Universal Robots URScript: fai_chun_2024_v2.script

def fai_chun_2024_v2():
  set_tcp(p[0.0,0.0,0.0,0.0,0.0,0.0])
  set_gravity([0.0, 0.0, 9.82])
  set_target_payload(1.070000, [0.002000, 0.003000, 0.057000], [0.001723, 0.001723, 0.001723, 0.000000, 0.000000, 0.000000])
  set_tool_communication(True, 1000000, 2, 1, 1.5, 3.5)
  set_tool_output_mode(0)
  set_tool_digital_output_mode(0, 1)
  set_tool_digital_output_mode(1, 1)
  set_tool_voltage(0)
  step_count_453dca7f_7b0c_4a5f_b250_0e1aac3a1e4a = 0.0
  thread Step_Counter_Thread_f9e71c20_d700_42f0_a2ea_6ea405c4239a():
    while (True):
      step_count_453dca7f_7b0c_4a5f_b250_0e1aac3a1e4a = step_count_453dca7f_7b0c_4a5f_b250_0e1aac3a1e4a + 1.0
      sync()
    end
  end
  run Step_Counter_Thread_f9e71c20_d700_42f0_a2ea_6ea405c4239a()
  set_safety_mode_transition_hardness(1)
  set_standard_analog_input_domain(0, 1)
  set_standard_analog_input_domain(1, 1)
  set_tool_analog_input_domain(0, 1)
  set_tool_analog_input_domain(1, 1)
  set_analog_outputdomain(0, 0)
  set_analog_outputdomain(1, 0)
  set_input_actions_to_default()
  global Plane_1=p[-0.700006141123905,1.3454883874109249E-6,0.3910559577028425,-1.2089868272251132,-1.2089999932245832,1.20858562628424]
  global Plane_2=p[0.0,0.0,0.0,0.0,0.0,0.0]
  global Point_1=p[0.6913645118948067,-0.12399382748223003,0.49223711947071,-1.2983729986843258,1.1259514972191385,-1.2203503861141718]
  # begin: URCap Installation Node
  #   Source: External Control, 1.0.5, FZI Research Center for Information Technology
  #   Type: External Control
  # end: URCap Installation Node
  $ 1 "Robot Program"
  $ 2 "Script: test_first_drawing_8_m18.script"
  def Machining1():
    # Default parameters:
    global speed_ms = 0.3
    global speed_rads = 0.75
    global accel_mss = 3
    global accel_radss = 1.2
    global blend_radius_m = 0.001

    # Add subprograms here
    # Start of main program
    # Program generated by RoboDK v5.6.5 for UR10e on 02/02/2024 17:18:51
    # Using nominal kinematics.
    blend_radius_m = 0.001
    speed_ms = 1.000
    # set_reference(p[0.123734, -0.230000, -0.017586, 0.000000, 0.000000, 0.000000])
    set_tcp(p[0.000000, 0.000000, 0.252000, 0.000000, 0.000000, 0.000000])
    # Show Tool
    movej([-0.347318, -0.633716, -2.608659, -1.470014, 1.570796, 1.223478],accel_radss,speed_rads,0,blend_radius_m)
    movel([-0.347318, -0.633716, -2.608659, -1.470014, 1.570796, 1.223478],accel_mss,speed_ms,0,blend_radius_m)
    # Splitting Linear movement in 6 (instruction 7: MoveL 3)
    movel([-0.347318, -0.640193, -2.637183, -1.435013, 1.570796, 1.223478],accel_mss,speed_ms,0,blend_radius_m)
    movel([-0.347318, -0.649079, -2.665529, -1.397781, 1.570796, 1.223478],accel_mss,speed_ms,0,blend_radius_m)
    movel([-0.347318, -0.660784, -2.693691, -1.357914, 1.570796, 1.223478],accel_mss,speed_ms,0,blend_radius_m)
    movel([-0.347318, -0.675813, -2.721660, -1.314916, 1.570796, 1.223478],accel_mss,speed_ms,0,blend_radius_m)
    movel([-0.347318, -0.694799, -2.749422, -1.268169, 1.570796, 1.223478],accel_mss,speed_ms,0,blend_radius_m)
    movel([-0.347318, -0.718542, -2.776954, -1.216893, 1.570796, 1.223478],accel_mss,speed_ms,0,blend_radius_m)
    movel([-0.347318, -0.718542, -2.776954, -1.216893, 1.570796, 1.223478],accel_mss,speed_ms,0,blend_radius_m)
    speed_ms = 1.000
    movel([-0.347318, -0.718542, -2.776954, -1.216893, 1.570796, 1.223478],accel_mss,speed_ms,0,blend_radius_m)
    movel([-0.347318, -0.718542, -2.776954, -1.216893, 1.570796, 1.223478],accel_mss,speed_ms,0,blend_radius_m)
    movel([-0.347318, -0.718542, -2.776954, -1.216893, 1.570796, 1.223478],accel_mss,speed_ms,0,blend_radius_m)
    speed_ms = 0.005
    # Splitting Linear movement in 2 (instruction 14: MoveL 8)
    movel([-0.347318, -0.703674, -2.760464, -1.248252, 1.570796, 1.223478],accel_mss,speed_ms,0,blend_radius_m)
    movel([-0.347318, -0.690649, -2.743887, -1.277853, 1.570796, 1.223478],accel_mss,speed_ms,0,blend_radius_m)
    speed_ms = 1.000
    # Splitting Linear movement in 2 (instruction 16: MoveL 9)
    movel([-0.347318, -0.703674, -2.760464, -1.248252, 1.570796, 1.223478],accel_mss,speed_ms,0,blend_radius_m)
    movel([-0.347318, -0.718542, -2.776954, -1.216893, 1.570796, 1.223478],accel_mss,speed_ms,0,blend_radius_m)
    speed_ms = 0.040
    movel([-0.347318, -0.718542, -2.776954, -1.216893, 1.570796, 1.223478],accel_mss,speed_ms,0,blend_radius_m)
    speed_ms = 1.000
    movel([-0.347318, -0.718542, -2.776954, -1.216893, 1.570796, 1.223478],accel_mss,speed_ms,0,blend_radius_m)
    # Splitting Linear movement in 8 (instruction 21: MoveL 12)
    movel([-0.279547, -0.705399, -2.778747, -1.228243, 1.570796, 1.291249],accel_mss,speed_ms,0,blend_radius_m)
    movel([-0.214126, -0.697642, -2.779767, -1.234980, 1.570796, 1.356670],accel_mss,speed_ms,0,blend_radius_m)
    movel([-0.151686, -0.695510, -2.780043, -1.236837, 1.570796, 1.419111],accel_mss,speed_ms,0,blend_radius_m)
    movel([-0.092735, -0.699070, -2.779582, -1.233738, 1.570796, 1.478061],accel_mss,speed_ms,0,blend_radius_m)
    movel([-0.037636, -0.708211, -2.778371, -1.225808, 1.570796, 1.533160],accel_mss,speed_ms,0,blend_radius_m)
    movel([0.013408, -0.722651, -2.776377, -1.213361, 1.570796, 1.584204],accel_mss,speed_ms,0,blend_radius_m)
    movel([0.060342, -0.741966, -2.773553, -1.196870, 1.570796, 1.631138],accel_mss,speed_ms,0,blend_radius_m)
    movel([0.103238, -0.765618, -2.769843, -1.176929, 1.570796, 1.674034],accel_mss,speed_ms,0,blend_radius_m)
    speed_ms = 0.005
    movel([0.103238, -0.804647, -2.801882, -1.105860, 1.570796, 1.674034],accel_mss,speed_ms,0,blend_radius_m)
    speed_ms = 0.025
    movel([0.099003, -0.816037, -2.799931, -1.096421, 1.570796, 1.669799],accel_mss,speed_ms,0,blend_radius_m)
    movel([0.096673, -0.821763, -2.798925, -1.091701, 1.570796, 1.667470],accel_mss,speed_ms,0,blend_radius_m)
    movel([0.094160, -0.827491, -2.797901, -1.086997, 1.570796, 1.664957],accel_mss,speed_ms,0,blend_radius_m)
    movel([0.091439, -0.833203, -2.796862, -1.082324, 1.570796, 1.662235],accel_mss,speed_ms,0,blend_radius_m)
    movel([0.088481, -0.838881, -2.795812, -1.077696, 1.570796, 1.659277],accel_mss,speed_ms,0,blend_radius_m)
    movel([0.085256, -0.844515, -2.794752, -1.073122, 1.570796, 1.656052],accel_mss,speed_ms,0,blend_radius_m)
    movel([0.081733, -0.850085, -2.793687, -1.068617, 1.570796, 1.652529],accel_mss,speed_ms,0,blend_radius_m)
    movel([0.083042, -0.847657, -2.794154, -1.070579, 1.570796, 1.653838],accel_mss,speed_ms,0,blend_radius_m)
    movel([0.084251, -0.844625, -2.794731, -1.073032, 1.570796, 1.655047],accel_mss,speed_ms,0,blend_radius_m)
    movel([0.084988, -0.841795, -2.795266, -1.075328, 1.570796, 1.655784],accel_mss,speed_ms,0,blend_radius_m)
    movel([0.085056, -0.840717, -2.795468, -1.076203, 1.570796, 1.655853],accel_mss,speed_ms,0,blend_radius_m)
    movel([0.084865, -0.839997, -2.795603, -1.076788, 1.570796, 1.655661],accel_mss,speed_ms,0,blend_radius_m)
    movel([0.084363, -0.839721, -2.795655, -1.077013, 1.570796, 1.655159],accel_mss,speed_ms,0,blend_radius_m)
    movel([0.083642, -0.839986, -2.795605, -1.076798, 1.570796, 1.654438],accel_mss,speed_ms,0,blend_radius_m)
    movel([0.082745, -0.840716, -2.795469, -1.076205, 1.570796, 1.653541],accel_mss,speed_ms,0,blend_radius_m)
    movel([0.081691, -0.841855, -2.795255, -1.075279, 1.570796, 1.652488],accel_mss,speed_ms,0,blend_radius_m)
    movel([0.079266, -0.845068, -2.794647, -1.072674, 1.570796, 1.650063],accel_mss,speed_ms,0,blend_radius_m)
    movel([0.076623, -0.849077, -2.793881, -1.069431, 1.570796, 1.647419],accel_mss,speed_ms,0,blend_radius_m)
    movel([0.071649, -0.857391, -2.792264, -1.062734, 1.570796, 1.642445],accel_mss,speed_ms,0,blend_radius_m)
    movel([0.068651, -0.862666, -2.791217, -1.058506, 1.570796, 1.639447],accel_mss,speed_ms,0,blend_radius_m)
    movel([0.064188, -0.870043, -2.789727, -1.052619, 1.570796, 1.634984],accel_mss,speed_ms,0,blend_radius_m)
    movel([0.061723, -0.873582, -2.789001, -1.049806, 1.570796, 1.632519],accel_mss,speed_ms,0,blend_radius_m)
    movel([0.059000, -0.876910, -2.788311, -1.047167, 1.570796, 1.629797],accel_mss,speed_ms,0,blend_radius_m)
    movel([0.059565, -0.875920, -2.788517, -1.047951, 1.570796, 1.630361],accel_mss,speed_ms,0,blend_radius_m)
    movel([0.059963, -0.874506, -2.788810, -1.049073, 1.570796, 1.630760],accel_mss,speed_ms,0,blend_radius_m)
    movel([0.060312, -0.871037, -2.789524, -1.051828, 1.570796, 1.631108],accel_mss,speed_ms,0,blend_radius_m)
    movel([0.060135, -0.867813, -2.790181, -1.054395, 1.570796, 1.630931],accel_mss,speed_ms,0,blend_radius_m)
    movel([0.059871, -0.866703, -2.790406, -1.055280, 1.570796, 1.630667],accel_mss,speed_ms,0,blend_radius_m)
    movel([0.059510, -0.866152, -2.790517, -1.055720, 1.570796, 1.630307],accel_mss,speed_ms,0,blend_radius_m)
    movel([0.058443, -0.865920, -2.790564, -1.055905, 1.570796, 1.629239],accel_mss,speed_ms,0,blend_radius_m)
    movel([0.057361, -0.866264, -2.790494, -1.055630, 1.570796, 1.628157],accel_mss,speed_ms,0,blend_radius_m)
    movel([0.056273, -0.867069, -2.790332, -1.054988, 1.570796, 1.627069],accel_mss,speed_ms,0,blend_radius_m)
    movel([0.055192, -0.868224, -2.790097, -1.054067, 1.570796, 1.625988],accel_mss,speed_ms,0,blend_radius_m)
    movel([0.053117, -0.871081, -2.789515, -1.051793, 1.570796, 1.623913],accel_mss,speed_ms,0,blend_radius_m)
    movel([0.051240, -0.873903, -2.788935, -1.049551, 1.570796, 1.622036],accel_mss,speed_ms,0,blend_radius_m)
    movel([0.048159, -0.878161, -2.788050, -1.046177, 1.570796, 1.618955],accel_mss,speed_ms,0,blend_radius_m)
    movel([0.045025, -0.882057, -2.787232, -1.043100, 1.570796, 1.615821],accel_mss,speed_ms,0,blend_radius_m)
    movel([0.041653, -0.885597, -2.786480, -1.040311, 1.570796, 1.612450],accel_mss,speed_ms,0,blend_radius_m)
    movel([0.037875, -0.888760, -2.785803, -1.037827, 1.570796, 1.608671],accel_mss,speed_ms,0,blend_radius_m)
    movel([0.039996, -0.885529, -2.786495, -1.040365, 1.570796, 1.610792],accel_mss,speed_ms,0,blend_radius_m)
    movel([0.041714, -0.882272, -2.787187, -1.042931, 1.570796, 1.612511],accel_mss,speed_ms,0,blend_radius_m)
    movel([0.042253, -0.880669, -2.787525, -1.044195, 1.570796, 1.613050],accel_mss,speed_ms,0,blend_radius_m)
    movel([0.042461, -0.879225, -2.787828, -1.045336, 1.570796, 1.613258],accel_mss,speed_ms,0,blend_radius_m)
    movel([0.042292, -0.878069, -2.788070, -1.046250, 1.570796, 1.613089],accel_mss,speed_ms,0,blend_radius_m)
    movel([0.041677, -0.877359, -2.788218, -1.046812, 1.570796, 1.612473],accel_mss,speed_ms,0,blend_radius_m)
    movel([0.040341, -0.877266, -2.788237, -1.046886, 1.570796, 1.611137],accel_mss,speed_ms,0,blend_radius_m)
    movel([0.038655, -0.877918, -2.788101, -1.046370, 1.570796, 1.609451],accel_mss,speed_ms,0,blend_radius_m)
    movel([0.036784, -0.879064, -2.787862, -1.045463, 1.570796, 1.607581],accel_mss,speed_ms,0,blend_radius_m)
    movel([0.034907, -0.880432, -2.787574, -1.044382, 1.570796, 1.605704],accel_mss,speed_ms,0,blend_radius_m)
    speed_ms = 0.005
    movel([0.034907, -0.871171, -2.781452, -1.059766, 1.570796, 1.605704],accel_mss,speed_ms,0,blend_radius_m)
    speed_ms = 0.040
    movel([0.039187, -0.905585, -2.773922, -1.032882, 1.570796, 1.609983],accel_mss,speed_ms,0,blend_radius_m)
    speed_ms = 0.005
    movel([0.039187, -0.915087, -2.779923, -1.017379, 1.570796, 1.609983],accel_mss,speed_ms,0,blend_radius_m)
    speed_ms = 0.025
    movel([0.040063, -0.912485, -2.780523, -1.019380, 1.570796, 1.610860],accel_mss,speed_ms,0,blend_radius_m)
    movel([0.041212, -0.909802, -2.781138, -1.021449, 1.570796, 1.612008],accel_mss,speed_ms,0,blend_radius_m)
    movel([0.042603, -0.907086, -2.781756, -1.023548, 1.570796, 1.613399],accel_mss,speed_ms,0,blend_radius_m)
    movel([0.044220, -0.904367, -2.782369, -1.025653, 1.570796, 1.615016],accel_mss,speed_ms,0,blend_radius_m)
    movel([0.046036, -0.901683, -2.782970, -1.027736, 1.570796, 1.616833],accel_mss,speed_ms,0,blend_radius_m)
    movel([0.048030, -0.899079, -2.783549, -1.029761, 1.570796, 1.618826],accel_mss,speed_ms,0,blend_radius_m)
    movel([0.050173, -0.896594, -2.784098, -1.031697, 1.570796, 1.620970],accel_mss,speed_ms,0,blend_radius_m)
    movel([0.052448, -0.894262, -2.784609, -1.033518, 1.570796, 1.623244],accel_mss,speed_ms,0,blend_radius_m)
    movel([0.055966, -0.891152, -2.785286, -1.035951, 1.570796, 1.626763],accel_mss,speed_ms,0,blend_radius_m)
    movel([0.059406, -0.888643, -2.785828, -1.037918, 1.570796, 1.630203],accel_mss,speed_ms,0,blend_radius_m)
    movel([0.062755, -0.886700, -2.786245, -1.039444, 1.570796, 1.633551],accel_mss,speed_ms,0,blend_radius_m)
    movel([0.065992, -0.885289, -2.786546, -1.040553, 1.570796, 1.636789],accel_mss,speed_ms,0,blend_radius_m)
    movel([0.069107, -0.884376, -2.786741, -1.041273, 1.570796, 1.639903],accel_mss,speed_ms,0,blend_radius_m)
    movel([0.072089, -0.883921, -2.786837, -1.041631, 1.570796, 1.642886],accel_mss,speed_ms,0,blend_radius_m)
    movel([0.074921, -0.883892, -2.786843, -1.041654, 1.570796, 1.645718],accel_mss,speed_ms,0,blend_radius_m)
    movel([0.077596, -0.884243, -2.786769, -1.041377, 1.570796, 1.648392],accel_mss,speed_ms,0,blend_radius_m)
    movel([0.080100, -0.884937, -2.786621, -1.040831, 1.570796, 1.650897],accel_mss,speed_ms,0,blend_radius_m)
    movel([0.082429, -0.885929, -2.786410, -1.040050, 1.570796, 1.653226],accel_mss,speed_ms,0,blend_radius_m)
    movel([0.086527, -0.888639, -2.785829, -1.037921, 1.570796, 1.657323],accel_mss,speed_ms,0,blend_radius_m)
    movel([0.089831, -0.892019, -2.785098, -1.035272, 1.570796, 1.660627],accel_mss,speed_ms,0,blend_radius_m)
    movel([0.092285, -0.895737, -2.784286, -1.032366, 1.570796, 1.663082],accel_mss,speed_ms,0,blend_radius_m)
    movel([0.094271, -0.900108, -2.783321, -1.028960, 1.570796, 1.665068],accel_mss,speed_ms,0,blend_radius_m)
    movel([0.095818, -0.904870, -2.782256, -1.025263, 1.570796, 1.666614],accel_mss,speed_ms,0,blend_radius_m)
    movel([0.096977, -0.909954, -2.781103, -1.021331, 1.570796, 1.667773],accel_mss,speed_ms,0,blend_radius_m)
    movel([0.097796, -0.915302, -2.779873, -1.017214, 1.570796, 1.668593],accel_mss,speed_ms,0,blend_radius_m)
    movel([0.098327, -0.920849, -2.778578, -1.012961, 1.570796, 1.669123],accel_mss,speed_ms,0,blend_radius_m)
    movel([0.098623, -0.926536, -2.777231, -1.008623, 1.570796, 1.669419],accel_mss,speed_ms,0,blend_radius_m)
    movel([0.098699, -0.938097, -2.774425, -0.999867, 1.570796, 1.669496],accel_mss,speed_ms,0,blend_radius_m)
    movel([0.098679, -0.946146, -2.772420, -0.993823, 1.570796, 1.669475],accel_mss,speed_ms,0,blend_radius_m)
    movel([0.098990, -0.949904, -2.771469, -0.991016, 1.570796, 1.669787],accel_mss,speed_ms,0,blend_radius_m)
    movel([0.099728, -0.953315, -2.770597, -0.988477, 1.570796, 1.670524],accel_mss,speed_ms,0,blend_radius_m)
    movel([0.101334, -0.957271, -2.769576, -0.985542, 1.570796, 1.672130],accel_mss,speed_ms,0,blend_radius_m)
    movel([0.102938, -0.961235, -2.768543, -0.982611, 1.570796, 1.673734],accel_mss,speed_ms,0,blend_radius_m)
    movel([0.103450, -0.963372, -2.767981, -0.981036, 1.570796, 1.674246],accel_mss,speed_ms,0,blend_radius_m)
    movel([0.103612, -0.965694, -2.767367, -0.979328, 1.570796, 1.674408],accel_mss,speed_ms,0,blend_radius_m)
    movel([0.103314, -0.968251, -2.766686, -0.977452, 1.570796, 1.674110],accel_mss,speed_ms,0,blend_radius_m)
    movel([0.102446, -0.971104, -2.765921, -0.975363, 1.570796, 1.673242],accel_mss,speed_ms,0,blend_radius_m)
    movel([0.105204, -0.963895, -2.767843, -0.980651, 1.570796, 1.676000],accel_mss,speed_ms,0,blend_radius_m)
    movel([0.107656, -0.956738, -2.769715, -0.985937, 1.570796, 1.678453],accel_mss,speed_ms,0,blend_radius_m)
    movel([0.112022, -0.942382, -2.773363, -0.996644, 1.570796, 1.682818],accel_mss,speed_ms,0,blend_radius_m)
    movel([0.114252, -0.934348, -2.775344, -1.002696, 1.570796, 1.685049],accel_mss,speed_ms,0,blend_radius_m)
    movel([0.116303, -0.926313, -2.777284, -1.008792, 1.570796, 1.687099],accel_mss,speed_ms,0,blend_radius_m)
    movel([0.120000, -0.910186, -2.781050, -1.021153, 1.570796, 1.690796],accel_mss,speed_ms,0,blend_radius_m)
    movel([0.123189, -0.894316, -2.784597, -1.033475, 1.570796, 1.693985],accel_mss,speed_ms,0,blend_radius_m)
    movel([0.124444, -0.886431, -2.786302, -1.039655, 1.570796, 1.695240],accel_mss,speed_ms,0,blend_radius_m)
    movel([0.125300, -0.878768, -2.787924, -1.045698, 1.570796, 1.696096],accel_mss,speed_ms,0,blend_radius_m)
    movel([0.125558, -0.872961, -2.789129, -1.050299, 1.570796, 1.696354],accel_mss,speed_ms,0,blend_radius_m)
    movel([0.125550, -0.867277, -2.790290, -1.054823, 1.570796, 1.696346],accel_mss,speed_ms,0,blend_radius_m)
    movel([0.125564, -0.861512, -2.791448, -1.059429, 1.570796, 1.696360],accel_mss,speed_ms,0,blend_radius_m)
    movel([0.125892, -0.855463, -2.792642, -1.064283, 1.570796, 1.696688],accel_mss,speed_ms,0,blend_radius_m)
    movel([0.126174, -0.853732, -2.792980, -1.065676, 1.570796, 1.696971],accel_mss,speed_ms,0,blend_radius_m)
    movel([0.126768, -0.851845, -2.793347, -1.067197, 1.570796, 1.697564],accel_mss,speed_ms,0,blend_radius_m)
    movel([0.127727, -0.850055, -2.793693, -1.068641, 1.570796, 1.698523],accel_mss,speed_ms,0,blend_radius_m)
    movel([0.128369, -0.849267, -2.793845, -1.069277, 1.570796, 1.699165],accel_mss,speed_ms,0,blend_radius_m)
    movel([0.129128, -0.848589, -2.793975, -1.069825, 1.570796, 1.699924],accel_mss,speed_ms,0,blend_radius_m)
    movel([0.130203, -0.847993, -2.794089, -1.070307, 1.570796, 1.700999],accel_mss,speed_ms,0,blend_radius_m)
    movel([0.131205, -0.847692, -2.794147, -1.070550, 1.570796, 1.702002],accel_mss,speed_ms,0,blend_radius_m)
    movel([0.136443, -0.846800, -2.794317, -1.071272, 1.570796, 1.707239],accel_mss,speed_ms,0,blend_radius_m)
    movel([0.141107, -0.846730, -2.794331, -1.071328, 1.570796, 1.711903],accel_mss,speed_ms,0,blend_radius_m)
    movel([0.145236, -0.847408, -2.794201, -1.070780, 1.570796, 1.716033],accel_mss,speed_ms,0,blend_radius_m)
    movel([0.148868, -0.848777, -2.793939, -1.069673, 1.570796, 1.719664],accel_mss,speed_ms,0,blend_radius_m)
    movel([0.152040, -0.850763, -2.793556, -1.068069, 1.570796, 1.722836],accel_mss,speed_ms,0,blend_radius_m)
    movel([0.154794, -0.853295, -2.793066, -1.066029, 1.570796, 1.725591],accel_mss,speed_ms,0,blend_radius_m)
    movel([0.157172, -0.856303, -2.792478, -1.063608, 1.570796, 1.727968],accel_mss,speed_ms,0,blend_radius_m)
    movel([0.159211, -0.859725, -2.791803, -1.060862, 1.570796, 1.730008],accel_mss,speed_ms,0,blend_radius_m)
    movel([0.160959, -0.863485, -2.791054, -1.057851, 1.570796, 1.731755],accel_mss,speed_ms,0,blend_radius_m)
    movel([0.162459, -0.867515, -2.790241, -1.054633, 1.570796, 1.733256],accel_mss,speed_ms,0,blend_radius_m)
    movel([0.164883, -0.876120, -2.788476, -1.047793, 1.570796, 1.735679],accel_mss,speed_ms,0,blend_radius_m)
    movel([0.168591, -0.893763, -2.784718, -1.033908, 1.570796, 1.739387],accel_mss,speed_ms,0,blend_radius_m)
    movel([0.169326, -0.896378, -2.784145, -1.031866, 1.570796, 1.740123],accel_mss,speed_ms,0,blend_radius_m)
    movel([0.169951, -0.897409, -2.783918, -1.031062, 1.570796, 1.740747],accel_mss,speed_ms,0,blend_radius_m)
    movel([0.170857, -0.898104, -2.783765, -1.030520, 1.570796, 1.741654],accel_mss,speed_ms,0,blend_radius_m)
    movel([0.172730, -0.898342, -2.783712, -1.030335, 1.570796, 1.743527],accel_mss,speed_ms,0,blend_radius_m)
    movel([0.173763, -0.898109, -2.783764, -1.030517, 1.570796, 1.744559],accel_mss,speed_ms,0,blend_radius_m)
    movel([0.174848, -0.897661, -2.783863, -1.030865, 1.570796, 1.745644],accel_mss,speed_ms,0,blend_radius_m)
    movel([0.177114, -0.896234, -2.784177, -1.031978, 1.570796, 1.747911],accel_mss,speed_ms,0,blend_radius_m)
    movel([0.179442, -0.894230, -2.784616, -1.033543, 1.570796, 1.750238],accel_mss,speed_ms,0,blend_radius_m)
    movel([0.181730, -0.891828, -2.785139, -1.035421, 1.570796, 1.752527],accel_mss,speed_ms,0,blend_radius_m)
    movel([0.183885, -0.889205, -2.785707, -1.037477, 1.570796, 1.754681],accel_mss,speed_ms,0,blend_radius_m)
    movel([0.185811, -0.886530, -2.786281, -1.039578, 1.570796, 1.756607],accel_mss,speed_ms,0,blend_radius_m)
    movel([0.187395, -0.883990, -2.786823, -1.041576, 1.570796, 1.758191],accel_mss,speed_ms,0,blend_radius_m)
    movel([0.189829, -0.879607, -2.787748, -1.045035, 1.570796, 1.760625],accel_mss,speed_ms,0,blend_radius_m)
    movel([0.192128, -0.875169, -2.788673, -1.048547, 1.570796, 1.762924],accel_mss,speed_ms,0,blend_radius_m)
    movel([0.196297, -0.866208, -2.790506, -1.055675, 1.570796, 1.767093],accel_mss,speed_ms,0,blend_radius_m)
    movel([0.199888, -0.857253, -2.792291, -1.062845, 1.570796, 1.770685],accel_mss,speed_ms,0,blend_radius_m)
    movel([0.202872, -0.848454, -2.794001, -1.069934, 1.570796, 1.773668],accel_mss,speed_ms,0,blend_radius_m)
    movel([0.203890, -0.845164, -2.794629, -1.072596, 1.570796, 1.774687],accel_mss,speed_ms,0,blend_radius_m)
    movel([0.205148, -0.841814, -2.795262, -1.075312, 1.570796, 1.775945],accel_mss,speed_ms,0,blend_radius_m)
    movel([0.205967, -0.840137, -2.795577, -1.076675, 1.570796, 1.776764],accel_mss,speed_ms,0,blend_radius_m)
    movel([0.206968, -0.838457, -2.795891, -1.078041, 1.570796, 1.777765],accel_mss,speed_ms,0,blend_radius_m)
    movel([0.208190, -0.836788, -2.796201, -1.079400, 1.570796, 1.778986],accel_mss,speed_ms,0,blend_radius_m)
    movel([0.209672, -0.835140, -2.796506, -1.080743, 1.570796, 1.780468],accel_mss,speed_ms,0,blend_radius_m)
    movel([0.211828, -0.833391, -2.796827, -1.082170, 1.570796, 1.782624],accel_mss,speed_ms,0,blend_radius_m)
    movel([0.213930, -0.832412, -2.797007, -1.082970, 1.570796, 1.784726],accel_mss,speed_ms,0,blend_radius_m)
    movel([0.215839, -0.832117, -2.797061, -1.083211, 1.570796, 1.786635],accel_mss,speed_ms,0,blend_radius_m)
    movel([0.217434, -0.832412, -2.797007, -1.082970, 1.570796, 1.788230],accel_mss,speed_ms,0,blend_radius_m)
    movel([0.219614, -0.833608, -2.796788, -1.081993, 1.570796, 1.790410],accel_mss,speed_ms,0,blend_radius_m)
    movel([0.221498, -0.835247, -2.796486, -1.080656, 1.570796, 1.792294],accel_mss,speed_ms,0,blend_radius_m)
    movel([0.224602, -0.839257, -2.795742, -1.077390, 1.570796, 1.795398],accel_mss,speed_ms,0,blend_radius_m)
    movel([0.225793, -0.841420, -2.795336, -1.075632, 1.570796, 1.796589],accel_mss,speed_ms,0,blend_radius_m)
    movel([0.226689, -0.843790, -2.794890, -1.073710, 1.570796, 1.797485],accel_mss,speed_ms,0,blend_radius_m)
    movel([0.227311, -0.846341, -2.794405, -1.071643, 1.570796, 1.798107],accel_mss,speed_ms,0,blend_radius_m)
    movel([0.227671, -0.849068, -2.793883, -1.069438, 1.570796, 1.798467],accel_mss,speed_ms,0,blend_radius_m)
    movel([0.227787, -0.851949, -2.793327, -1.067113, 1.570796, 1.798583],accel_mss,speed_ms,0,blend_radius_m)
    movel([0.227345, -0.858132, -2.792118, -1.062139, 1.570796, 1.798141],accel_mss,speed_ms,0,blend_radius_m)
    movel([0.226817, -0.861403, -2.791470, -1.059517, 1.570796, 1.797613],accel_mss,speed_ms,0,blend_radius_m)
    movel([0.225239, -0.868228, -2.790097, -1.054065, 1.570796, 1.796035],accel_mss,speed_ms,0,blend_radius_m)
    movel([0.223056, -0.875348, -2.788636, -1.048405, 1.570796, 1.793852],accel_mss,speed_ms,0,blend_radius_m)
    movel([0.220382, -0.882670, -2.787102, -1.042617, 1.570796, 1.791179],accel_mss,speed_ms,0,blend_radius_m)
    movel([0.217344, -0.890081, -2.785518, -1.036790, 1.570796, 1.788140],accel_mss,speed_ms,0,blend_radius_m)
    movel([0.212440, -0.900905, -2.783144, -1.028340, 1.570796, 1.783236],accel_mss,speed_ms,0,blend_radius_m)
    movel([0.209759, -0.906300, -2.781933, -1.024155, 1.570796, 1.780555],accel_mss,speed_ms,0,blend_radius_m)
    movel([0.206897, -0.911655, -2.780714, -1.020020, 1.570796, 1.777694],accel_mss,speed_ms,0,blend_radius_m)
    movel([0.203841, -0.916936, -2.779494, -1.015959, 1.570796, 1.774638],accel_mss,speed_ms,0,blend_radius_m)
    movel([0.200578, -0.922122, -2.778279, -1.011988, 1.570796, 1.771374],accel_mss,speed_ms,0,blend_radius_m)
    movel([0.197078, -0.927198, -2.777072, -1.008119, 1.570796, 1.767874],accel_mss,speed_ms,0,blend_radius_m)
    movel([0.193334, -0.932132, -2.775884, -1.004374, 1.570796, 1.764130],accel_mss,speed_ms,0,blend_radius_m)
    movel([0.187774, -0.938770, -2.774259, -0.999360, 1.570796, 1.758571],accel_mss,speed_ms,0,blend_radius_m)
    movel([0.184722, -0.942091, -2.773435, -0.996862, 1.570796, 1.755518],accel_mss,speed_ms,0,blend_radius_m)
    movel([0.181561, -0.945236, -2.772649, -0.994504, 1.570796, 1.752357],accel_mss,speed_ms,0,blend_radius_m)
    movel([0.178351, -0.948070, -2.771934, -0.992385, 1.570796, 1.749147],accel_mss,speed_ms,0,blend_radius_m)
    movel([0.175145, -0.950463, -2.771326, -0.990600, 1.570796, 1.745942],accel_mss,speed_ms,0,blend_radius_m)
    movel([0.171998, -0.952282, -2.770862, -0.989245, 1.570796, 1.742794],accel_mss,speed_ms,0,blend_radius_m)
    movel([0.170463, -0.952939, -2.770693, -0.988756, 1.570796, 1.741259],accel_mss,speed_ms,0,blend_radius_m)
    movel([0.168966, -0.953400, -2.770575, -0.988414, 1.570796, 1.739762],accel_mss,speed_ms,0,blend_radius_m)
    movel([0.167355, -0.953668, -2.770506, -0.988215, 1.570796, 1.738151],accel_mss,speed_ms,0,blend_radius_m)
    movel([0.165897, -0.953659, -2.770509, -0.988221, 1.570796, 1.736693],accel_mss,speed_ms,0,blend_radius_m)
    movel([0.164579, -0.953403, -2.770574, -0.988411, 1.570796, 1.735376],accel_mss,speed_ms,0,blend_radius_m)
    movel([0.163394, -0.952918, -2.770699, -0.988772, 1.570796, 1.734191],accel_mss,speed_ms,0,blend_radius_m)
    movel([0.161377, -0.951372, -2.771095, -0.989923, 1.570796, 1.732173],accel_mss,speed_ms,0,blend_radius_m)
    movel([0.159776, -0.949206, -2.771646, -0.991537, 1.570796, 1.730573],accel_mss,speed_ms,0,blend_radius_m)
    movel([0.158515, -0.946621, -2.772300, -0.993467, 1.570796, 1.729312],accel_mss,speed_ms,0,blend_radius_m)
    movel([0.157523, -0.943813, -2.773006, -0.995571, 1.570796, 1.728319],accel_mss,speed_ms,0,blend_radius_m)
    movel([0.156059, -0.938308, -2.774373, -0.999708, 1.570796, 1.726855],accel_mss,speed_ms,0,blend_radius_m)
    movel([0.155407, -0.935714, -2.775011, -1.001664, 1.570796, 1.726203],accel_mss,speed_ms,0,blend_radius_m)
    movel([0.154469, -0.933401, -2.775575, -1.003413, 1.570796, 1.725266],accel_mss,speed_ms,0,blend_radius_m)
    movel([0.153768, -0.932521, -2.775789, -1.004079, 1.570796, 1.724565],accel_mss,speed_ms,0,blend_radius_m)
    movel([0.152844, -0.931916, -2.775936, -1.004537, 1.570796, 1.723640],accel_mss,speed_ms,0,blend_radius_m)
    movel([0.151650, -0.931657, -2.775999, -1.004733, 1.570796, 1.722446],accel_mss,speed_ms,0,blend_radius_m)
    movel([0.150136, -0.931808, -2.775962, -1.004619, 1.570796, 1.720932],accel_mss,speed_ms,0,blend_radius_m)
    movel([0.150460, -0.931850, -2.775952, -1.004587, 1.570796, 1.721256],accel_mss,speed_ms,0,blend_radius_m)
    movel([0.150631, -0.932144, -2.775881, -1.004364, 1.570796, 1.721428],accel_mss,speed_ms,0,blend_radius_m)
    movel([0.150538, -0.933432, -2.775568, -1.003389, 1.570796, 1.721335],accel_mss,speed_ms,0,blend_radius_m)
    movel([0.149924, -0.935541, -2.775053, -1.001795, 1.570796, 1.720720],accel_mss,speed_ms,0,blend_radius_m)
    movel([0.148873, -0.938338, -2.774366, -0.999685, 1.570796, 1.719669],accel_mss,speed_ms,0,blend_radius_m)
    movel([0.145761, -0.945454, -2.772594, -0.994341, 1.570796, 1.716558],accel_mss,speed_ms,0,blend_radius_m)
    movel([0.141805, -0.953724, -2.770492, -0.988173, 1.570796, 1.712601],accel_mss,speed_ms,0,blend_radius_m)
    movel([0.133669, -0.969714, -2.766295, -0.976380, 1.570796, 1.704466],accel_mss,speed_ms,0,blend_radius_m)
    movel([0.128816, -0.978712, -2.763854, -0.969823, 1.570796, 1.699612],accel_mss,speed_ms,0,blend_radius_m)
    movel([0.123189, -0.987937, -2.761291, -0.963161, 1.570796, 1.693985],accel_mss,speed_ms,0,blend_radius_m)
    movel([0.117520, -0.996914, -2.758737, -0.956737, 1.570796, 1.688317],accel_mss,speed_ms,0,blend_radius_m)
    movel([0.111784, -1.005734, -2.756170, -0.950484, 1.570796, 1.682581],accel_mss,speed_ms,0,blend_radius_m)
    movel([0.100475, -1.022487, -2.751131, -0.938772, 1.570796, 1.671271],accel_mss,speed_ms,0,blend_radius_m)
    movel([0.094794, -1.030269, -2.748715, -0.933405, 1.570796, 1.665590],accel_mss,speed_ms,0,blend_radius_m)
    movel([0.091825, -1.033997, -2.747541, -0.930851, 1.570796, 1.662621],accel_mss,speed_ms,0,blend_radius_m)
    movel([0.088750, -1.037576, -2.746404, -0.928409, 1.570796, 1.659547],accel_mss,speed_ms,0,blend_radius_m)
    movel([0.085541, -1.040978, -2.745313, -0.926098, 1.570796, 1.656337],accel_mss,speed_ms,0,blend_radius_m)
    movel([0.082188, -1.044173, -2.744280, -0.923936, 1.570796, 1.652984],accel_mss,speed_ms,0,blend_radius_m)
    movel([0.083080, -1.037857, -2.746314, -0.928218, 1.570796, 1.653877],accel_mss,speed_ms,0,blend_radius_m)
    movel([0.083098, -1.036102, -2.746873, -0.929413, 1.570796, 1.653894],accel_mss,speed_ms,0,blend_radius_m)
    movel([0.082806, -1.035506, -2.747063, -0.929820, 1.570796, 1.653602],accel_mss,speed_ms,0,blend_radius_m)
    movel([0.082192, -1.035305, -2.747127, -0.929958, 1.570796, 1.652988],accel_mss,speed_ms,0,blend_radius_m)
    movel([0.081500, -1.035506, -2.747063, -0.929820, 1.570796, 1.652296],accel_mss,speed_ms,0,blend_radius_m)
    movel([0.080757, -1.035964, -2.746917, -0.929508, 1.570796, 1.651553],accel_mss,speed_ms,0,blend_radius_m)
    movel([0.077209, -1.038847, -2.745997, -0.927545, 1.570796, 1.648006],accel_mss,speed_ms,0,blend_radius_m)
    movel([0.075121, -1.040203, -2.745562, -0.926624, 1.570796, 1.645918],accel_mss,speed_ms,0,blend_radius_m)
    movel([0.073038, -1.041260, -2.745222, -0.925907, 1.570796, 1.643835],accel_mss,speed_ms,0,blend_radius_m)
    movel([0.071014, -1.041990, -2.744987, -0.925413, 1.570796, 1.641811],accel_mss,speed_ms,0,blend_radius_m)
    movel([0.070412, -1.042035, -2.744972, -0.925382, 1.570796, 1.641209],accel_mss,speed_ms,0,blend_radius_m)
    movel([0.070248, -1.041684, -2.745085, -0.925620, 1.570796, 1.641045],accel_mss,speed_ms,0,blend_radius_m)
    movel([0.070851, -1.039778, -2.745699, -0.926912, 1.570796, 1.641647],accel_mss,speed_ms,0,blend_radius_m)
    movel([0.070805, -1.039231, -2.745874, -0.927284, 1.570796, 1.641602],accel_mss,speed_ms,0,blend_radius_m)
    movel([0.070484, -1.038915, -2.745976, -0.927499, 1.570796, 1.641280],accel_mss,speed_ms,0,blend_radius_m)
    movel([0.069972, -1.038824, -2.746005, -0.927560, 1.570796, 1.640769],accel_mss,speed_ms,0,blend_radius_m)
    movel([0.069354, -1.038956, -2.745962, -0.927470, 1.570796, 1.640150],accel_mss,speed_ms,0,blend_radius_m)
    movel([0.068039, -1.039712, -2.745720, -0.926957, 1.570796, 1.638835],accel_mss,speed_ms,0,blend_radius_m)
    movel([0.058760, -1.047544, -2.743181, -0.921664, 1.570796, 1.629557],accel_mss,speed_ms,0,blend_radius_m)
    movel([0.061502, -1.044730, -2.744099, -0.923560, 1.570796, 1.632298],accel_mss,speed_ms,0,blend_radius_m)
    movel([0.064208, -1.041708, -2.745077, -0.925603, 1.570796, 1.635005],accel_mss,speed_ms,0,blend_radius_m)
    movel([0.066855, -1.038528, -2.746099, -0.927762, 1.570796, 1.637652],accel_mss,speed_ms,0,blend_radius_m)
    movel([0.069434, -1.035223, -2.747153, -0.930013, 1.570796, 1.640231],accel_mss,speed_ms,0,blend_radius_m)
    movel([0.074318, -1.028404, -2.749299, -0.934686, 1.570796, 1.645115],accel_mss,speed_ms,0,blend_radius_m)
    movel([0.078717, -1.021600, -2.751403, -0.939386, 1.570796, 1.649514],accel_mss,speed_ms,0,blend_radius_m)
    movel([0.083218, -1.014129, -2.753672, -0.944588, 1.570796, 1.654015],accel_mss,speed_ms,0,blend_radius_m)
    movel([0.087522, -1.006495, -2.755946, -0.949948, 1.570796, 1.658318],accel_mss,speed_ms,0,blend_radius_m)
    movel([0.089529, -1.002639, -2.757078, -0.952672, 1.570796, 1.660325],accel_mss,speed_ms,0,blend_radius_m)
    movel([0.091408, -0.998767, -2.758203, -0.955419, 1.570796, 1.662204],accel_mss,speed_ms,0,blend_radius_m)
    movel([0.093124, -0.994896, -2.759317, -0.958176, 1.570796, 1.663920],accel_mss,speed_ms,0,blend_radius_m)
    movel([0.094652, -0.991026, -2.760419, -0.960944, 1.570796, 1.665448],accel_mss,speed_ms,0,blend_radius_m)
    movel([0.095451, -0.988640, -2.761093, -0.962656, 1.570796, 1.666247],accel_mss,speed_ms,0,blend_radius_m)
    movel([0.096078, -0.986282, -2.761755, -0.964351, 1.570796, 1.666874],accel_mss,speed_ms,0,blend_radius_m)
    movel([0.096856, -0.981679, -2.763036, -0.967674, 1.570796, 1.667652],accel_mss,speed_ms,0,blend_radius_m)
    movel([0.097044, -0.977274, -2.764248, -0.970867, 1.570796, 1.667841],accel_mss,speed_ms,0,blend_radius_m)
    movel([0.096698, -0.973122, -2.765377, -0.973890, 1.570796, 1.667494],accel_mss,speed_ms,0,blend_radius_m)
    movel([0.095885, -0.969272, -2.766413, -0.976704, 1.570796, 1.666682],accel_mss,speed_ms,0,blend_radius_m)
    movel([0.094673, -0.965779, -2.767344, -0.979266, 1.570796, 1.665469],accel_mss,speed_ms,0,blend_radius_m)
    movel([0.093117, -0.962698, -2.768158, -0.981533, 1.570796, 1.663914],accel_mss,speed_ms,0,blend_radius_m)
    movel([0.091294, -0.960075, -2.768846, -0.983468, 1.570796, 1.662090],accel_mss,speed_ms,0,blend_radius_m)
    movel([0.089890, -0.959016, -2.769122, -0.984250, 1.570796, 1.660686],accel_mss,speed_ms,0,blend_radius_m)
    movel([0.088130, -0.958709, -2.769202, -0.984477, 1.570796, 1.658926],accel_mss,speed_ms,0,blend_radius_m)
    movel([0.086122, -0.959094, -2.769102, -0.984192, 1.570796, 1.656919],accel_mss,speed_ms,0,blend_radius_m)
    movel([0.083982, -0.960110, -2.768837, -0.983442, 1.570796, 1.654778],accel_mss,speed_ms,0,blend_radius_m)
    movel([0.081811, -0.961688, -2.768424, -0.982277, 1.570796, 1.652607],accel_mss,speed_ms,0,blend_radius_m)
    movel([0.079718, -0.963766, -2.767877, -0.980746, 1.570796, 1.650515],accel_mss,speed_ms,0,blend_radius_m)
    movel([0.077822, -0.966270, -2.767214, -0.978906, 1.570796, 1.648618],accel_mss,speed_ms,0,blend_radius_m)
    movel([0.076220, -0.969132, -2.766451, -0.976806, 1.570796, 1.647017],accel_mss,speed_ms,0,blend_radius_m)
    movel([0.074089, -0.973507, -2.765273, -0.973609, 1.570796, 1.644885],accel_mss,speed_ms,0,blend_radius_m)
    movel([0.071800, -0.977835, -2.764094, -0.970460, 1.570796, 1.642596],accel_mss,speed_ms,0,blend_radius_m)
    movel([0.069334, -0.982081, -2.762925, -0.967383, 1.570796, 1.640130],accel_mss,speed_ms,0,blend_radius_m)
    movel([0.066663, -0.986220, -2.761773, -0.964397, 1.570796, 1.637459],accel_mss,speed_ms,0,blend_radius_m)
    movel([0.063776, -0.990214, -2.760649, -0.961526, 1.570796, 1.634573],accel_mss,speed_ms,0,blend_radius_m)
    movel([0.060645, -0.994040, -2.759562, -0.958788, 1.570796, 1.631441],accel_mss,speed_ms,0,blend_radius_m)
    movel([0.057249, -0.997671, -2.758520, -0.956199, 1.570796, 1.628045],accel_mss,speed_ms,0,blend_radius_m)
    movel([0.053570, -1.001076, -2.757533, -0.953780, 1.570796, 1.624366],accel_mss,speed_ms,0,blend_radius_m)
    movel([0.051576, -1.002632, -2.757080, -0.952677, 1.570796, 1.622373],accel_mss,speed_ms,0,blend_radius_m)
    movel([0.049554, -1.003954, -2.756693, -0.951742, 1.570796, 1.620351],accel_mss,speed_ms,0,blend_radius_m)
    movel([0.045495, -1.006165, -2.756043, -0.950181, 1.570796, 1.616291],accel_mss,speed_ms,0,blend_radius_m)
    movel([0.042339, -1.007580, -2.755625, -0.949184, 1.570796, 1.613135],accel_mss,speed_ms,0,blend_radius_m)
    movel([0.039357, -1.008537, -2.755342, -0.948510, 1.570796, 1.610153],accel_mss,speed_ms,0,blend_radius_m)
    movel([0.036547, -1.009071, -2.755184, -0.948135, 1.570796, 1.607343],accel_mss,speed_ms,0,blend_radius_m)
    movel([0.033898, -1.009219, -2.755140, -0.948031, 1.570796, 1.604694],accel_mss,speed_ms,0,blend_radius_m)
    movel([0.031401, -1.009020, -2.755199, -0.948170, 1.570796, 1.602198],accel_mss,speed_ms,0,blend_radius_m)
    movel([0.029051, -1.008506, -2.755351, -0.948532, 1.570796, 1.599847],accel_mss,speed_ms,0,blend_radius_m)
    movel([0.026847, -1.007705, -2.755589, -0.949096, 1.570796, 1.597643],accel_mss,speed_ms,0,blend_radius_m)
    movel([0.024781, -1.006657, -2.755898, -0.949834, 1.570796, 1.595577],accel_mss,speed_ms,0,blend_radius_m)
    movel([0.022847, -1.005395, -2.756270, -0.950724, 1.570796, 1.593644],accel_mss,speed_ms,0,blend_radius_m)
    movel([0.021045, -1.003943, -2.756696, -0.951750, 1.570796, 1.591841],accel_mss,speed_ms,0,blend_radius_m)
    movel([0.017815, -1.000626, -2.757664, -0.954099, 1.570796, 1.588611],accel_mss,speed_ms,0,blend_radius_m)
    movel([0.015062, -0.996962, -2.758724, -0.956703, 1.570796, 1.585858],accel_mss,speed_ms,0,blend_radius_m)
    movel([0.012764, -0.993221, -2.759795, -0.959373, 1.570796, 1.583560],accel_mss,speed_ms,0,blend_radius_m)
    movel([0.011207, -0.990175, -2.760660, -0.961554, 1.570796, 1.582003],accel_mss,speed_ms,0,blend_radius_m)
    movel([0.009810, -0.986850, -2.761596, -0.963943, 1.570796, 1.580607],accel_mss,speed_ms,0,blend_radius_m)
    movel([0.008595, -0.983255, -2.762599, -0.966534, 1.570796, 1.579392],accel_mss,speed_ms,0,blend_radius_m)
    movel([0.007599, -0.979403, -2.763664, -0.969322, 1.570796, 1.578395],accel_mss,speed_ms,0,blend_radius_m)
    movel([0.006839, -0.975307, -2.764784, -0.972297, 1.570796, 1.577636],accel_mss,speed_ms,0,blend_radius_m)
    movel([0.006352, -0.970979, -2.765955, -0.975455, 1.570796, 1.577148],accel_mss,speed_ms,0,blend_radius_m)
    movel([0.006169, -0.966426, -2.767172, -0.978790, 1.570796, 1.576965],accel_mss,speed_ms,0,blend_radius_m)
    movel([0.006319, -0.961661, -2.768431, -0.982297, 1.570796, 1.577116],accel_mss,speed_ms,0,blend_radius_m)
    movel([0.006833, -0.956691, -2.769726, -0.985971, 1.570796, 1.577629],accel_mss,speed_ms,0,blend_radius_m)
    movel([0.007743, -0.951537, -2.771052, -0.989800, 1.570796, 1.578539],accel_mss,speed_ms,0,blend_radius_m)
    movel([0.009082, -0.946198, -2.772407, -0.993784, 1.570796, 1.579879],accel_mss,speed_ms,0,blend_radius_m)
    movel([0.010890, -0.940689, -2.773784, -0.997916, 1.570796, 1.581686],accel_mss,speed_ms,0,blend_radius_m)
    movel([0.013194, -0.935026, -2.775179, -1.002184, 1.570796, 1.583990],accel_mss,speed_ms,0,blend_radius_m)
    movel([0.016036, -0.929212, -2.776589, -1.006588, 1.570796, 1.586832],accel_mss,speed_ms,0,blend_radius_m)
    movel([0.019444, -0.923275, -2.778006, -1.011108, 1.570796, 1.590241],accel_mss,speed_ms,0,blend_radius_m)
    movel([0.023456, -0.917223, -2.779427, -1.015739, 1.570796, 1.594252],accel_mss,speed_ms,0,blend_radius_m)
    movel([0.025200, -0.914937, -2.779958, -1.017494, 1.570796, 1.595997],accel_mss,speed_ms,0,blend_radius_m)
    movel([0.026159, -0.913903, -2.780197, -1.018289, 1.570796, 1.596955],accel_mss,speed_ms,0,blend_radius_m)
    movel([0.027177, -0.913030, -2.780398, -1.018961, 1.570796, 1.597974],accel_mss,speed_ms,0,blend_radius_m)
    movel([0.028707, -0.912202, -2.780589, -1.019599, 1.570796, 1.599504],accel_mss,speed_ms,0,blend_radius_m)
    movel([0.030067, -0.911980, -2.780640, -1.019770, 1.570796, 1.600863],accel_mss,speed_ms,0,blend_radius_m)
    movel([0.031201, -0.912261, -2.780575, -1.019553, 1.570796, 1.601998],accel_mss,speed_ms,0,blend_radius_m)
    movel([0.032055, -0.912941, -2.780419, -1.019030, 1.570796, 1.602852],accel_mss,speed_ms,0,blend_radius_m)
    movel([0.033252, -0.915181, -2.779901, -1.017307, 1.570796, 1.604048],accel_mss,speed_ms,0,blend_radius_m)
    movel([0.033894, -0.917978, -2.779251, -1.015160, 1.570796, 1.604690],accel_mss,speed_ms,0,blend_radius_m)
    movel([0.034569, -0.924025, -2.777828, -1.010536, 1.570796, 1.605365],accel_mss,speed_ms,0,blend_radius_m)
    movel([0.034987, -0.924952, -2.777608, -1.009829, 1.570796, 1.605784],accel_mss,speed_ms,0,blend_radius_m)
    movel([0.035456, -0.924977, -2.777602, -1.009810, 1.570796, 1.606252],accel_mss,speed_ms,0,blend_radius_m)
    movel([0.036179, -0.924616, -2.777688, -1.010085, 1.570796, 1.606975],accel_mss,speed_ms,0,blend_radius_m)
    movel([0.037373, -0.921722, -2.778373, -1.012294, 1.570796, 1.608169],accel_mss,speed_ms,0,blend_radius_m)
    movel([0.038411, -0.918803, -2.779058, -1.014528, 1.570796, 1.609208],accel_mss,speed_ms,0,blend_radius_m)
    movel([0.039032, -0.927882, -2.776908, -1.007598, 1.570796, 1.609828],accel_mss,speed_ms,0,blend_radius_m)
    movel([0.039969, -0.936638, -2.774784, -1.000967, 1.570796, 1.610765],accel_mss,speed_ms,0,blend_radius_m)
    movel([0.041215, -0.945072, -2.772690, -0.994627, 1.570796, 1.612011],accel_mss,speed_ms,0,blend_radius_m)
    movel([0.042760, -0.953194, -2.770628, -0.988567, 1.570796, 1.613556],accel_mss,speed_ms,0,blend_radius_m)
    movel([0.043563, -0.956609, -2.769748, -0.986032, 1.570796, 1.614359],accel_mss,speed_ms,0,blend_radius_m)
    movel([0.044726, -0.959899, -2.768892, -0.983598, 1.570796, 1.615523],accel_mss,speed_ms,0,blend_radius_m)
    movel([0.045510, -0.961348, -2.768513, -0.982528, 1.570796, 1.616307],accel_mss,speed_ms,0,blend_radius_m)
    movel([0.046464, -0.962585, -2.768188, -0.981616, 1.570796, 1.617260],accel_mss,speed_ms,0,blend_radius_m)
    movel([0.047618, -0.963547, -2.767935, -0.980907, 1.570796, 1.618414],accel_mss,speed_ms,0,blend_radius_m)
    movel([0.049000, -0.964172, -2.767770, -0.980447, 1.570796, 1.619796],accel_mss,speed_ms,0,blend_radius_m)
    movel([0.050105, -0.964362, -2.767719, -0.980308, 1.570796, 1.620902],accel_mss,speed_ms,0,blend_radius_m)
    movel([0.052567, -0.964071, -2.767796, -0.980522, 1.570796, 1.623364],accel_mss,speed_ms,0,blend_radius_m)
    movel([0.053899, -0.963624, -2.767914, -0.980851, 1.570796, 1.624696],accel_mss,speed_ms,0,blend_radius_m)
    movel([0.056704, -0.962221, -2.768284, -0.981885, 1.570796, 1.627500],accel_mss,speed_ms,0,blend_radius_m)
    movel([0.059623, -0.960242, -2.768802, -0.983344, 1.570796, 1.630419],accel_mss,speed_ms,0,blend_radius_m)
    movel([0.062557, -0.957835, -2.769430, -0.985124, 1.570796, 1.633353],accel_mss,speed_ms,0,blend_radius_m)
    movel([0.065410, -0.955126, -2.770131, -0.987132, 1.570796, 1.636207],accel_mss,speed_ms,0,blend_radius_m)
    movel([0.068084, -0.952261, -2.770867, -0.989261, 1.570796, 1.638880],accel_mss,speed_ms,0,blend_radius_m)
    movel([0.070469, -0.949382, -2.771601, -0.991405, 1.570796, 1.641266],accel_mss,speed_ms,0,blend_radius_m)
    speed_ms = 0.005
    movel([0.070469, -0.939687, -2.765727, -1.006974, 1.570796, 1.641266],accel_mss,speed_ms,0,blend_radius_m)
    speed_ms = 0.040
    movel([0.057022, -0.948626, -2.763452, -1.000310, 1.570796, 1.627819],accel_mss,speed_ms,0,blend_radius_m)
    speed_ms = 0.005
    movel([0.057022, -0.958365, -2.769292, -0.984732, 1.570796, 1.627819],accel_mss,speed_ms,0,blend_radius_m)
    speed_ms = 0.025
    movel([0.058920, -0.955968, -2.769914, -0.986507, 1.570796, 1.629716],accel_mss,speed_ms,0,blend_radius_m)
    movel([0.062572, -0.950701, -2.771266, -0.990422, 1.570796, 1.633368],accel_mss,speed_ms,0,blend_radius_m)
    movel([0.064292, -0.947886, -2.771981, -0.992522, 1.570796, 1.635088],accel_mss,speed_ms,0,blend_radius_m)
    movel([0.067440, -0.942037, -2.773449, -0.996903, 1.570796, 1.638237],accel_mss,speed_ms,0,blend_radius_m)
    movel([0.070101, -0.936077, -2.774922, -1.001390, 1.570796, 1.640897],accel_mss,speed_ms,0,blend_radius_m)
    movel([0.071205, -0.933134, -2.775640, -1.003615, 1.570796, 1.642002],accel_mss,speed_ms,0,blend_radius_m)
    movel([0.072133, -0.930250, -2.776339, -1.005801, 1.570796, 1.642930],accel_mss,speed_ms,0,blend_radius_m)
    movel([0.073394, -0.924802, -2.777644, -1.009944, 1.570796, 1.644191],accel_mss,speed_ms,0,blend_radius_m)
    movel([0.073696, -0.922294, -2.778238, -1.011857, 1.570796, 1.644492],accel_mss,speed_ms,0,blend_radius_m)
    movel([0.073747, -0.919983, -2.778782, -1.013624, 1.570796, 1.644544],accel_mss,speed_ms,0,blend_radius_m)
    movel([0.073537, -0.917894, -2.779271, -1.015224, 1.570796, 1.644333],accel_mss,speed_ms,0,blend_radius_m)
    movel([0.073044, -0.916061, -2.779697, -1.016631, 1.570796, 1.643840],accel_mss,speed_ms,0,blend_radius_m)
    movel([0.072118, -0.914083, -2.780155, -1.018151, 1.570796, 1.642914],accel_mss,speed_ms,0,blend_radius_m)
    movel([0.070922, -0.912398, -2.780543, -1.019447, 1.570796, 1.641719],accel_mss,speed_ms,0,blend_radius_m)
    movel([0.069439, -0.911090, -2.780844, -1.020456, 1.570796, 1.640235],accel_mss,speed_ms,0,blend_radius_m)
    movel([0.067653, -0.910244, -2.781037, -1.021108, 1.570796, 1.638450],accel_mss,speed_ms,0,blend_radius_m)
    movel([0.065548, -0.909941, -2.781106, -1.021342, 1.570796, 1.636344],accel_mss,speed_ms,0,blend_radius_m)
    movel([0.063115, -0.910264, -2.781033, -1.021093, 1.570796, 1.633912],accel_mss,speed_ms,0,blend_radius_m)
    movel([0.060342, -0.911293, -2.780797, -1.020299, 1.570796, 1.631138],accel_mss,speed_ms,0,blend_radius_m)
    movel([0.057220, -0.913096, -2.780383, -1.018910, 1.570796, 1.628016],accel_mss,speed_ms,0,blend_radius_m)
    movel([0.055065, -0.914732, -2.780005, -1.017652, 1.570796, 1.625861],accel_mss,speed_ms,0,blend_radius_m)
    movel([0.052968, -0.916674, -2.779555, -1.016160, 1.570796, 1.623764],accel_mss,speed_ms,0,blend_radius_m)
    movel([0.051000, -0.918838, -2.779050, -1.014501, 1.570796, 1.621797],accel_mss,speed_ms,0,blend_radius_m)
    movel([0.049221, -0.921151, -2.778507, -1.012731, 1.570796, 1.620018],accel_mss,speed_ms,0,blend_radius_m)
    movel([0.047692, -0.923535, -2.777944, -1.010909, 1.570796, 1.618488],accel_mss,speed_ms,0,blend_radius_m)
    movel([0.046474, -0.925917, -2.777378, -1.009094, 1.570796, 1.617270],accel_mss,speed_ms,0,blend_radius_m)
    movel([0.045629, -0.928219, -2.776828, -1.007343, 1.570796, 1.616426],accel_mss,speed_ms,0,blend_radius_m)
    movel([0.045209, -0.930375, -2.776309, -1.005705, 1.570796, 1.616006],accel_mss,speed_ms,0,blend_radius_m)
    speed_ms = 0.005
    movel([0.045209, -0.920782, -2.770363, -1.021244, 1.570796, 1.616006],accel_mss,speed_ms,0,blend_radius_m)
    speed_ms = 0.040
    # Splitting Linear movement in 2 (instruction 399: MoveL 378)
    movel([0.099245, -0.926509, -2.768984, -1.016896, 1.570796, 1.670041],accel_mss,speed_ms,0,blend_radius_m)
    movel([0.150339, -0.936625, -2.766494, -1.009270, 1.570796, 1.721135],accel_mss,speed_ms,0,blend_radius_m)
    speed_ms = 0.005
    movel([0.150339, -0.946305, -2.772380, -0.993704, 1.570796, 1.721135],accel_mss,speed_ms,0,blend_radius_m)
    speed_ms = 0.025
    movel([0.148401, -0.957492, -2.769519, -0.985378, 1.570796, 1.719197],accel_mss,speed_ms,0,blend_radius_m)
    movel([0.147061, -0.963170, -2.768034, -0.981185, 1.570796, 1.717857],accel_mss,speed_ms,0,blend_radius_m)
    movel([0.146164, -0.966105, -2.767258, -0.979026, 1.570796, 1.716960],accel_mss,speed_ms,0,blend_radius_m)
    movel([0.145065, -0.969126, -2.766452, -0.976811, 1.570796, 1.715861],accel_mss,speed_ms,0,blend_radius_m)
    movel([0.143636, -0.972379, -2.765578, -0.974432, 1.570796, 1.714432],accel_mss,speed_ms,0,blend_radius_m)
    movel([0.142756, -0.973992, -2.765141, -0.973255, 1.570796, 1.713552],accel_mss,speed_ms,0,blend_radius_m)
    movel([0.141713, -0.975571, -2.764712, -0.972105, 1.570796, 1.712509],accel_mss,speed_ms,0,blend_radius_m)
    movel([0.141774, -0.973142, -2.765372, -0.973875, 1.570796, 1.712570],accel_mss,speed_ms,0,blend_radius_m)
    movel([0.141427, -0.970989, -2.765952, -0.975448, 1.570796, 1.712223],accel_mss,speed_ms,0,blend_radius_m)
    movel([0.141070, -0.970464, -2.766093, -0.975831, 1.570796, 1.711867],accel_mss,speed_ms,0,blend_radius_m)
    movel([0.140680, -0.970519, -2.766079, -0.975791, 1.570796, 1.711476],accel_mss,speed_ms,0,blend_radius_m)
    movel([0.140225, -0.970790, -2.766006, -0.975593, 1.570796, 1.711021],accel_mss,speed_ms,0,blend_radius_m)
    movel([0.139306, -0.971693, -2.765763, -0.974933, 1.570796, 1.710103],accel_mss,speed_ms,0,blend_radius_m)
    movel([0.138016, -0.973402, -2.765301, -0.973686, 1.570796, 1.708813],accel_mss,speed_ms,0,blend_radius_m)
    movel([0.136990, -0.975107, -2.764839, -0.972443, 1.570796, 1.707786],accel_mss,speed_ms,0,blend_radius_m)
    movel([0.136178, -0.976802, -2.764377, -0.971210, 1.570796, 1.706974],accel_mss,speed_ms,0,blend_radius_m)
    movel([0.135533, -0.978483, -2.763917, -0.969989, 1.570796, 1.706329],accel_mss,speed_ms,0,blend_radius_m)
    movel([0.133609, -0.985092, -2.762088, -0.965209, 1.570796, 1.704405],accel_mss,speed_ms,0,blend_radius_m)
    movel([0.132293, -0.988998, -2.760992, -0.962399, 1.570796, 1.703090],accel_mss,speed_ms,0,blend_radius_m)
    movel([0.130743, -0.992936, -2.759876, -0.959577, 1.570796, 1.701539],accel_mss,speed_ms,0,blend_radius_m)
    movel([0.128897, -0.996890, -2.758744, -0.956755, 1.570796, 1.699693],accel_mss,speed_ms,0,blend_radius_m)
    movel([0.126697, -1.000825, -2.757606, -0.953957, 1.570796, 1.697493],accel_mss,speed_ms,0,blend_radius_m)
    movel([0.127358, -0.997907, -2.758451, -0.956030, 1.570796, 1.698155],accel_mss,speed_ms,0,blend_radius_m)
    movel([0.127362, -0.995316, -2.759197, -0.957877, 1.570796, 1.698159],accel_mss,speed_ms,0,blend_radius_m)
    movel([0.127215, -0.994759, -2.759356, -0.958274, 1.570796, 1.698012],accel_mss,speed_ms,0,blend_radius_m)
    movel([0.126834, -0.994458, -2.759442, -0.958489, 1.570796, 1.697630],accel_mss,speed_ms,0,blend_radius_m)
    movel([0.126328, -0.994556, -2.759414, -0.958419, 1.570796, 1.697124],accel_mss,speed_ms,0,blend_radius_m)
    movel([0.125751, -0.994918, -2.759310, -0.958161, 1.570796, 1.696547],accel_mss,speed_ms,0,blend_radius_m)
    movel([0.124623, -0.996050, -2.758986, -0.957353, 1.570796, 1.695420],accel_mss,speed_ms,0,blend_radius_m)
    movel([0.123414, -0.997670, -2.758520, -0.956199, 1.570796, 1.694211],accel_mss,speed_ms,0,blend_radius_m)
    movel([0.122379, -0.999349, -2.758034, -0.955005, 1.570796, 1.693175],accel_mss,speed_ms,0,blend_radius_m)
    movel([0.120699, -1.002791, -2.757033, -0.952565, 1.570796, 1.691495],accel_mss,speed_ms,0,blend_radius_m)
    movel([0.117931, -1.009559, -2.755039, -0.947792, 1.570796, 1.688728],accel_mss,speed_ms,0,blend_radius_m)
    movel([0.116127, -1.013330, -2.753912, -0.945147, 1.570796, 1.686924],accel_mss,speed_ms,0,blend_radius_m)
    movel([0.114102, -1.017081, -2.752781, -0.942528, 1.570796, 1.684899],accel_mss,speed_ms,0,blend_radius_m)
    movel([0.111806, -1.020760, -2.751660, -0.939969, 1.570796, 1.682603],accel_mss,speed_ms,0,blend_radius_m)
    movel([0.109193, -1.024322, -2.750565, -0.937502, 1.570796, 1.679989],accel_mss,speed_ms,0,blend_radius_m)
    movel([0.109726, -1.022715, -2.751060, -0.938613, 1.570796, 1.680522],accel_mss,speed_ms,0,blend_radius_m)
    movel([0.110248, -1.019701, -2.751984, -0.940704, 1.570796, 1.681044],accel_mss,speed_ms,0,blend_radius_m)
    movel([0.110227, -1.018338, -2.752399, -0.941652, 1.570796, 1.681023],accel_mss,speed_ms,0,blend_radius_m)
    movel([0.110067, -1.017806, -2.752561, -0.942023, 1.570796, 1.680864],accel_mss,speed_ms,0,blend_radius_m)
    movel([0.109596, -1.017704, -2.752591, -0.942093, 1.570796, 1.680393],accel_mss,speed_ms,0,blend_radius_m)
    movel([0.108907, -1.018257, -2.752424, -0.941709, 1.570796, 1.679704],accel_mss,speed_ms,0,blend_radius_m)
    movel([0.107358, -1.020006, -2.751890, -0.940492, 1.570796, 1.678155],accel_mss,speed_ms,0,blend_radius_m)
    movel([0.106015, -1.021782, -2.751347, -0.939260, 1.570796, 1.676811],accel_mss,speed_ms,0,blend_radius_m)
    movel([0.103706, -1.025395, -2.750234, -0.936761, 1.570796, 1.674502],accel_mss,speed_ms,0,blend_radius_m)
    movel([0.101492, -1.029036, -2.749101, -0.934252, 1.570796, 1.672288],accel_mss,speed_ms,0,blend_radius_m)
    movel([0.100268, -1.030853, -2.748532, -0.933004, 1.570796, 1.671065],accel_mss,speed_ms,0,blend_radius_m)
    movel([0.098885, -1.032662, -2.747963, -0.931764, 1.570796, 1.669682],accel_mss,speed_ms,0,blend_radius_m)
    movel([0.095286, -1.036857, -2.746633, -0.928899, 1.570796, 1.666082],accel_mss,speed_ms,0,blend_radius_m)
    movel([0.091564, -1.040897, -2.745339, -0.926153, 1.570796, 1.662361],accel_mss,speed_ms,0,blend_radius_m)
    movel([0.087758, -1.044788, -2.744080, -0.923521, 1.570796, 1.658554],accel_mss,speed_ms,0,blend_radius_m)
    movel([0.083896, -1.048550, -2.742851, -0.920988, 1.570796, 1.654693],accel_mss,speed_ms,0,blend_radius_m)
    speed_ms = 0.005
    movel([0.083896, -1.038544, -2.737374, -0.936471, 1.570796, 1.654693],accel_mss,speed_ms,0,blend_radius_m)
    speed_ms = 0.040
    movel([0.054600, -1.009438, -2.746481, -0.956470, 1.570796, 1.625396],accel_mss,speed_ms,0,blend_radius_m)
    speed_ms = 0.005
    movel([0.054600, -1.019390, -2.752078, -0.940920, 1.570796, 1.625396],accel_mss,speed_ms,0,blend_radius_m)
    speed_ms = 0.025
    movel([0.055801, -1.017946, -2.752518, -0.941925, 1.570796, 1.626598],accel_mss,speed_ms,0,blend_radius_m)
    movel([0.056876, -1.016380, -2.752993, -0.943016, 1.570796, 1.627672],accel_mss,speed_ms,0,blend_radius_m)
    movel([0.058812, -1.013014, -2.754007, -0.945368, 1.570796, 1.629608],accel_mss,speed_ms,0,blend_radius_m)
    movel([0.060727, -1.009568, -2.755036, -0.947785, 1.570796, 1.631523],accel_mss,speed_ms,0,blend_radius_m)
    movel([0.061780, -1.007898, -2.755531, -0.948960, 1.570796, 1.632577],accel_mss,speed_ms,0,blend_radius_m)
    movel([0.062951, -1.006312, -2.756000, -0.950077, 1.570796, 1.633747],accel_mss,speed_ms,0,blend_radius_m)
    movel([0.063886, -1.005256, -2.756311, -0.950822, 1.570796, 1.634682],accel_mss,speed_ms,0,blend_radius_m)
    movel([0.064662, -1.004576, -2.756511, -0.951303, 1.570796, 1.635458],accel_mss,speed_ms,0,blend_radius_m)
    movel([0.065292, -1.004228, -2.756613, -0.951548, 1.570796, 1.636089],accel_mss,speed_ms,0,blend_radius_m)
    movel([0.065794, -1.004172, -2.756629, -0.951588, 1.570796, 1.636591],accel_mss,speed_ms,0,blend_radius_m)
    movel([0.066450, -1.004804, -2.756444, -0.951141, 1.570796, 1.637246],accel_mss,speed_ms,0,blend_radius_m)
    movel([0.066736, -1.006154, -2.756046, -0.950189, 1.570796, 1.637532],accel_mss,speed_ms,0,blend_radius_m)
    movel([0.066611, -1.009783, -2.754972, -0.947634, 1.570796, 1.637407],accel_mss,speed_ms,0,blend_radius_m)
    movel([0.066271, -1.012600, -2.754131, -0.945658, 1.570796, 1.637068],accel_mss,speed_ms,0,blend_radius_m)
    movel([0.068407, -1.009156, -2.755158, -0.948075, 1.570796, 1.639203],accel_mss,speed_ms,0,blend_radius_m)
    movel([0.070028, -1.005867, -2.756131, -0.950391, 1.570796, 1.640824],accel_mss,speed_ms,0,blend_radius_m)
    movel([0.071269, -1.002680, -2.757066, -0.952644, 1.570796, 1.642065],accel_mss,speed_ms,0,blend_radius_m)
    movel([0.072249, -0.999558, -2.757974, -0.954857, 1.570796, 1.643046],accel_mss,speed_ms,0,blend_radius_m)
    movel([0.074930, -0.990092, -2.760683, -0.961613, 1.570796, 1.645726],accel_mss,speed_ms,0,blend_radius_m)
    movel([0.076171, -0.986741, -2.761627, -0.964021, 1.570796, 1.646967],accel_mss,speed_ms,0,blend_radius_m)
    movel([0.076865, -0.985369, -2.762011, -0.965009, 1.570796, 1.647661],accel_mss,speed_ms,0,blend_radius_m)
    movel([0.077578, -0.984475, -2.762260, -0.965654, 1.570796, 1.648374],accel_mss,speed_ms,0,blend_radius_m)
    movel([0.078285, -0.983991, -2.762395, -0.966003, 1.570796, 1.649082],accel_mss,speed_ms,0,blend_radius_m)
    movel([0.078957, -0.983859, -2.762432, -0.966098, 1.570796, 1.649753],accel_mss,speed_ms,0,blend_radius_m)
    movel([0.079570, -0.984007, -2.762390, -0.965992, 1.570796, 1.650366],accel_mss,speed_ms,0,blend_radius_m)
    movel([0.080093, -0.984373, -2.762288, -0.965727, 1.570796, 1.650889],accel_mss,speed_ms,0,blend_radius_m)
    movel([0.080776, -0.985490, -2.761977, -0.964922, 1.570796, 1.651572],accel_mss,speed_ms,0,blend_radius_m)
    movel([0.080916, -0.987002, -2.761554, -0.963834, 1.570796, 1.651713],accel_mss,speed_ms,0,blend_radius_m)
    movel([0.080750, -0.989111, -2.760960, -0.962317, 1.570796, 1.651546],accel_mss,speed_ms,0,blend_radius_m)
    movel([0.080188, -0.993110, -2.759827, -0.959452, 1.570796, 1.650984],accel_mss,speed_ms,0,blend_radius_m)
    movel([0.082393, -0.986555, -2.761679, -0.964155, 1.570796, 1.653190],accel_mss,speed_ms,0,blend_radius_m)
    movel([0.083234, -0.983343, -2.762575, -0.966471, 1.570796, 1.654030],accel_mss,speed_ms,0,blend_radius_m)
    movel([0.084371, -0.977107, -2.764294, -0.970989, 1.570796, 1.655167],accel_mss,speed_ms,0,blend_radius_m)
    movel([0.084656, -0.974115, -2.765108, -0.973166, 1.570796, 1.655453],accel_mss,speed_ms,0,blend_radius_m)
    movel([0.084649, -0.968449, -2.766633, -0.977306, 1.570796, 1.655445],accel_mss,speed_ms,0,blend_radius_m)
    speed_ms = 0.005
    movel([0.084649, -0.958666, -2.760832, -0.992891, 1.570796, 1.655445],accel_mss,speed_ms,0,blend_radius_m)
    speed_ms = 0.040
    movel([0.064704, -0.986643, -2.753157, -0.972589, 1.570796, 1.635501],accel_mss,speed_ms,0,blend_radius_m)
    speed_ms = 0.005
    movel([0.064704, -0.996531, -2.758848, -0.957010, 1.570796, 1.635501],accel_mss,speed_ms,0,blend_radius_m)
    speed_ms = 0.025
    movel([0.062199, -1.000485, -2.757705, -0.954199, 1.570796, 1.632996],accel_mss,speed_ms,0,blend_radius_m)
    movel([0.059916, -1.004456, -2.756546, -0.951387, 1.570796, 1.630712],accel_mss,speed_ms,0,blend_radius_m)
    movel([0.055504, -1.012348, -2.754206, -0.945835, 1.570796, 1.626301],accel_mss,speed_ms,0,blend_radius_m)
    movel([0.053094, -1.016253, -2.753031, -0.943105, 1.570796, 1.623890],accel_mss,speed_ms,0,blend_radius_m)
    movel([0.050426, -1.020043, -2.751879, -0.940466, 1.570796, 1.621222],accel_mss,speed_ms,0,blend_radius_m)
    movel([0.047473, -1.023573, -2.750796, -0.938020, 1.570796, 1.618269],accel_mss,speed_ms,0,blend_radius_m)
    movel([0.045884, -1.025194, -2.750296, -0.936899, 1.570796, 1.616680],accel_mss,speed_ms,0,blend_radius_m)
    movel([0.044215, -1.026696, -2.749830, -0.935863, 1.570796, 1.615012],accel_mss,speed_ms,0,blend_radius_m)
    movel([0.045435, -1.025355, -2.750246, -0.936788, 1.570796, 1.616232],accel_mss,speed_ms,0,blend_radius_m)
    movel([0.046709, -1.023433, -2.750840, -0.938117, 1.570796, 1.617505],accel_mss,speed_ms,0,blend_radius_m)
    movel([0.047891, -1.021198, -2.751526, -0.939665, 1.570796, 1.618688],accel_mss,speed_ms,0,blend_radius_m)
    movel([0.048815, -1.018935, -2.752217, -0.941237, 1.570796, 1.619612],accel_mss,speed_ms,0,blend_radius_m)
    movel([0.049327, -1.016919, -2.752829, -0.942640, 1.570796, 1.620124],accel_mss,speed_ms,0,blend_radius_m)
    movel([0.049374, -1.016101, -2.753077, -0.943211, 1.570796, 1.620171],accel_mss,speed_ms,0,blend_radius_m)
    movel([0.049259, -1.015449, -2.753274, -0.943666, 1.570796, 1.620056],accel_mss,speed_ms,0,blend_radius_m)
    movel([0.048962, -1.015002, -2.753409, -0.943978, 1.570796, 1.619758],accel_mss,speed_ms,0,blend_radius_m)
    movel([0.048456, -1.014801, -2.753470, -0.944119, 1.570796, 1.619252],accel_mss,speed_ms,0,blend_radius_m)
    movel([0.047731, -1.014875, -2.753447, -0.944067, 1.570796, 1.618527],accel_mss,speed_ms,0,blend_radius_m)
    movel([0.046757, -1.015264, -2.753330, -0.943795, 1.570796, 1.617553],accel_mss,speed_ms,0,blend_radius_m)
    movel([0.045191, -1.016374, -2.752994, -0.943020, 1.570796, 1.615987],accel_mss,speed_ms,0,blend_radius_m)
    movel([0.038754, -1.022336, -2.751177, -0.938876, 1.570796, 1.609550],accel_mss,speed_ms,0,blend_radius_m)
    movel([0.036003, -1.024600, -2.750479, -0.937309, 1.570796, 1.606800],accel_mss,speed_ms,0,blend_radius_m)
    movel([0.033182, -1.026692, -2.749831, -0.935866, 1.570796, 1.603978],accel_mss,speed_ms,0,blend_radius_m)
    movel([0.030377, -1.028497, -2.749270, -0.934623, 1.570796, 1.601174],accel_mss,speed_ms,0,blend_radius_m)
    movel([0.027677, -1.029889, -2.748834, -0.933666, 1.570796, 1.598473],accel_mss,speed_ms,0,blend_radius_m)
    movel([0.025162, -1.030753, -2.748563, -0.933072, 1.570796, 1.595959],accel_mss,speed_ms,0,blend_radius_m)
    movel([0.022922, -1.030961, -2.748498, -0.932929, 1.570796, 1.593719],accel_mss,speed_ms,0,blend_radius_m)
    movel([0.023640, -1.030782, -2.748555, -0.933053, 1.570796, 1.594436],accel_mss,speed_ms,0,blend_radius_m)
    movel([0.024584, -1.030222, -2.748730, -0.933437, 1.570796, 1.595380],accel_mss,speed_ms,0,blend_radius_m)
    movel([0.026850, -1.028354, -2.749314, -0.934721, 1.570796, 1.597646],accel_mss,speed_ms,0,blend_radius_m)
    movel([0.029076, -1.026144, -2.750001, -0.936243, 1.570796, 1.599873],accel_mss,speed_ms,0,blend_radius_m)
    movel([0.030610, -1.024392, -2.750544, -0.937453, 1.570796, 1.601407],accel_mss,speed_ms,0,blend_radius_m)
    movel([0.031512, -1.023059, -2.750955, -0.938375, 1.570796, 1.602309],accel_mss,speed_ms,0,blend_radius_m)
    movel([0.031850, -1.022183, -2.751224, -0.938982, 1.570796, 1.602646],accel_mss,speed_ms,0,blend_radius_m)
    movel([0.031713, -1.021694, -2.751374, -0.939321, 1.570796, 1.602509],accel_mss,speed_ms,0,blend_radius_m)
    movel([0.031205, -1.021518, -2.751428, -0.939443, 1.570796, 1.602001],accel_mss,speed_ms,0,blend_radius_m)
    movel([0.029480, -1.021814, -2.751337, -0.939237, 1.570796, 1.600276],accel_mss,speed_ms,0,blend_radius_m)
    movel([0.027480, -1.022487, -2.751130, -0.938771, 1.570796, 1.598276],accel_mss,speed_ms,0,blend_radius_m)
    movel([0.022935, -1.024013, -2.750661, -0.937715, 1.570796, 1.593731],accel_mss,speed_ms,0,blend_radius_m)
    movel([0.018415, -1.025144, -2.750311, -0.936934, 1.570796, 1.589211],accel_mss,speed_ms,0,blend_radius_m)
    movel([0.016284, -1.025418, -2.750227, -0.936745, 1.570796, 1.587080],accel_mss,speed_ms,0,blend_radius_m)
    movel([0.014302, -1.025418, -2.750227, -0.936745, 1.570796, 1.585099],accel_mss,speed_ms,0,blend_radius_m)
    movel([0.012520, -1.025084, -2.750330, -0.936975, 1.570796, 1.583316],accel_mss,speed_ms,0,blend_radius_m)
    movel([0.010985, -1.024357, -2.750554, -0.937477, 1.570796, 1.581781],accel_mss,speed_ms,0,blend_radius_m)
    movel([0.013694, -1.023418, -2.750844, -0.938127, 1.570796, 1.584490],accel_mss,speed_ms,0,blend_radius_m)
    movel([0.015180, -1.022580, -2.751102, -0.938707, 1.570796, 1.585976],accel_mss,speed_ms,0,blend_radius_m)
    movel([0.015840, -1.022039, -2.751268, -0.939082, 1.570796, 1.586637],accel_mss,speed_ms,0,blend_radius_m)
    movel([0.016405, -1.021399, -2.751464, -0.939526, 1.570796, 1.587201],accel_mss,speed_ms,0,blend_radius_m)
    movel([0.016637, -1.020915, -2.751613, -0.939861, 1.570796, 1.587433],accel_mss,speed_ms,0,blend_radius_m)
    movel([0.016607, -1.020482, -2.751745, -0.940162, 1.570796, 1.587403],accel_mss,speed_ms,0,blend_radius_m)
    movel([0.015903, -1.019755, -2.751967, -0.940666, 1.570796, 1.586699],accel_mss,speed_ms,0,blend_radius_m)
    movel([0.014533, -1.019200, -2.752136, -0.941053, 1.570796, 1.585329],accel_mss,speed_ms,0,blend_radius_m)
    movel([0.012751, -1.018786, -2.752263, -0.941340, 1.570796, 1.583548],accel_mss,speed_ms,0,blend_radius_m)
    movel([0.006500, -1.018024, -2.752494, -0.941870, 1.570796, 1.577296],accel_mss,speed_ms,0,blend_radius_m)
    movel([0.004236, -1.017381, -2.752690, -0.942319, 1.570796, 1.575032],accel_mss,speed_ms,0,blend_radius_m)
    movel([0.002193, -1.016412, -2.752983, -0.942994, 1.570796, 1.572989],accel_mss,speed_ms,0,blend_radius_m)
    movel([0.000505, -1.015024, -2.753402, -0.943962, 1.570796, 1.571301],accel_mss,speed_ms,0,blend_radius_m)
    movel([-0.000711, -1.013128, -2.753972, -0.945288, 1.570796, 1.570085],accel_mss,speed_ms,0,blend_radius_m)
    movel([0.001381, -1.013849, -2.753756, -0.944784, 1.570796, 1.572178],accel_mss,speed_ms,0,blend_radius_m)
    movel([0.002688, -1.013947, -2.753727, -0.944716, 1.570796, 1.573484],accel_mss,speed_ms,0,blend_radius_m)
    movel([0.003961, -1.013588, -2.753834, -0.944966, 1.570796, 1.574757],accel_mss,speed_ms,0,blend_radius_m)
    movel([0.005179, -1.012693, -2.754103, -0.945593, 1.570796, 1.575975],accel_mss,speed_ms,0,blend_radius_m)
    movel([0.005913, -1.011660, -2.754412, -0.946317, 1.570796, 1.576710],accel_mss,speed_ms,0,blend_radius_m)
    movel([0.006136, -1.010626, -2.754721, -0.947042, 1.570796, 1.576932],accel_mss,speed_ms,0,blend_radius_m)
    movel([0.005821, -1.009724, -2.754989, -0.947675, 1.570796, 1.576618],accel_mss,speed_ms,0,blend_radius_m)
    movel([0.003187, -1.005673, -2.756188, -0.950528, 1.570796, 1.573983],accel_mss,speed_ms,0,blend_radius_m)
    movel([0.001186, -1.001161, -2.757509, -0.953720, 1.570796, 1.571982],accel_mss,speed_ms,0,blend_radius_m)
    movel([0.000471, -0.998653, -2.758236, -0.955500, 1.570796, 1.571267],accel_mss,speed_ms,0,blend_radius_m)
    movel([-0.000032, -0.995939, -2.759018, -0.957433, 1.570796, 1.570765],accel_mss,speed_ms,0,blend_radius_m)
    movel([-0.000300, -0.992983, -2.759863, -0.959543, 1.570796, 1.570496],accel_mss,speed_ms,0,blend_radius_m)
    movel([-0.000317, -0.989754, -2.760779, -0.961856, 1.570796, 1.570479],accel_mss,speed_ms,0,blend_radius_m)
    speed_ms = 0.005
    movel([-0.000317, -0.979888, -2.755062, -0.977439, 1.570796, 1.570479],accel_mss,speed_ms,0,blend_radius_m)
    speed_ms = 0.040
    movel([-0.042918, -0.973011, -2.756967, -0.982411, 1.570796, 1.527878],accel_mss,speed_ms,0,blend_radius_m)
    speed_ms = 0.005
    movel([-0.042918, -0.982852, -2.762711, -0.966825, 1.570796, 1.527878],accel_mss,speed_ms,0,blend_radius_m)
    speed_ms = 0.025
    movel([-0.039460, -0.976945, -2.764338, -0.971106, 1.570796, 1.531336],accel_mss,speed_ms,0,blend_radius_m)
    movel([-0.036128, -0.970978, -2.765955, -0.975456, 1.570796, 1.534668],accel_mss,speed_ms,0,blend_radius_m)
    movel([-0.029770, -0.958831, -2.769171, -0.984387, 1.570796, 1.541026],accel_mss,speed_ms,0,blend_radius_m)
    movel([-0.023836, -0.946436, -2.772347, -0.993606, 1.570796, 1.546960],accel_mss,speed_ms,0,blend_radius_m)
    movel([-0.018344, -0.933832, -2.775470, -1.003086, 1.570796, 1.552452],accel_mss,speed_ms,0,blend_radius_m)
    movel([-0.013310, -0.921060, -2.778529, -1.012800, 1.570796, 1.557486],accel_mss,speed_ms,0,blend_radius_m)
    movel([-0.008757, -0.908170, -2.781510, -1.022710, 1.570796, 1.562039],accel_mss,speed_ms,0,blend_radius_m)
    movel([-0.004705, -0.895218, -2.784400, -1.032771, 1.570796, 1.566091],accel_mss,speed_ms,0,blend_radius_m)
    movel([-0.001178, -0.882254, -2.787190, -1.042944, 1.570796, 1.569618],accel_mss,speed_ms,0,blend_radius_m)
    movel([0.001795, -0.869355, -2.789868, -1.053167, 1.570796, 1.572591],accel_mss,speed_ms,0,blend_radius_m)
    movel([0.004187, -0.856583, -2.792423, -1.063383, 1.570796, 1.574983],accel_mss,speed_ms,0,blend_radius_m)
    movel([0.005964, -0.844018, -2.794846, -1.073524, 1.570796, 1.576760],accel_mss,speed_ms,0,blend_radius_m)
    movel([0.007091, -0.831743, -2.797129, -1.083517, 1.570796, 1.577887],accel_mss,speed_ms,0,blend_radius_m)
    movel([0.007545, -0.819830, -2.799267, -1.093292, 1.570796, 1.578342],accel_mss,speed_ms,0,blend_radius_m)
    movel([0.007280, -0.808384, -2.801249, -1.102756, 1.570796, 1.578077],accel_mss,speed_ms,0,blend_radius_m)
    movel([0.006268, -0.797494, -2.803072, -1.111822, 1.570796, 1.577064],accel_mss,speed_ms,0,blend_radius_m)
    movel([0.003537, -0.782144, -2.805539, -1.124706, 1.570796, 1.574334],accel_mss,speed_ms,0,blend_radius_m)
    movel([0.003479, -0.779260, -2.805989, -1.127139, 1.570796, 1.574275],accel_mss,speed_ms,0,blend_radius_m)
    movel([0.003942, -0.776000, -2.806493, -1.129896, 1.570796, 1.574738],accel_mss,speed_ms,0,blend_radius_m)
    movel([0.005330, -0.771081, -2.807244, -1.134064, 1.570796, 1.576126],accel_mss,speed_ms,0,blend_radius_m)
    movel([0.007063, -0.766969, -2.807862, -1.137557, 1.570796, 1.577859],accel_mss,speed_ms,0,blend_radius_m)
    movel([0.008040, -0.765205, -2.808125, -1.139059, 1.570796, 1.578837],accel_mss,speed_ms,0,blend_radius_m)
    movel([0.010190, -0.762210, -2.808568, -1.141612, 1.570796, 1.580986],accel_mss,speed_ms,0,blend_radius_m)
    movel([0.011341, -0.760978, -2.808748, -1.142662, 1.570796, 1.582138],accel_mss,speed_ms,0,blend_radius_m)
    movel([0.013784, -0.758994, -2.809038, -1.144357, 1.570796, 1.584580],accel_mss,speed_ms,0,blend_radius_m)
    movel([0.016352, -0.757610, -2.809239, -1.145540, 1.570796, 1.587149],accel_mss,speed_ms,0,blend_radius_m)
    movel([0.018992, -0.756773, -2.809360, -1.146256, 1.570796, 1.589788],accel_mss,speed_ms,0,blend_radius_m)
    movel([0.021654, -0.756426, -2.809410, -1.146552, 1.570796, 1.592451],accel_mss,speed_ms,0,blend_radius_m)
    movel([0.024281, -0.756506, -2.809399, -1.146484, 1.570796, 1.595077],accel_mss,speed_ms,0,blend_radius_m)
    movel([0.026825, -0.756956, -2.809334, -1.146099, 1.570796, 1.597622],accel_mss,speed_ms,0,blend_radius_m)
    movel([0.031453, -0.758697, -2.809081, -1.144611, 1.570796, 1.602249],accel_mss,speed_ms,0,blend_radius_m)
    movel([0.035152, -0.761133, -2.808726, -1.142530, 1.570796, 1.605948],accel_mss,speed_ms,0,blend_radius_m)
    movel([0.037569, -0.763703, -2.808348, -1.140338, 1.570796, 1.608365],accel_mss,speed_ms,0,blend_radius_m)
    movel([0.039685, -0.767468, -2.807788, -1.137134, 1.570796, 1.610481],accel_mss,speed_ms,0,blend_radius_m)
    movel([0.041391, -0.771668, -2.807155, -1.133566, 1.570796, 1.612187],accel_mss,speed_ms,0,blend_radius_m)
    movel([0.043967, -0.780889, -2.805735, -1.125765, 1.570796, 1.614763],accel_mss,speed_ms,0,blend_radius_m)
    movel([0.046072, -0.790466, -2.804216, -1.117707, 1.570796, 1.616868],accel_mss,speed_ms,0,blend_radius_m)
    movel([0.048443, -0.799552, -2.802732, -1.110104, 1.570796, 1.619240],accel_mss,speed_ms,0,blend_radius_m)
    movel([0.051148, -0.807077, -2.801471, -1.103841, 1.570796, 1.621945],accel_mss,speed_ms,0,blend_radius_m)
    movel([0.052930, -0.810355, -2.800913, -1.101121, 1.570796, 1.623726],accel_mss,speed_ms,0,blend_radius_m)
    movel([0.055234, -0.813022, -2.800454, -1.098912, 1.570796, 1.626030],accel_mss,speed_ms,0,blend_radius_m)
    movel([0.056620, -0.813880, -2.800306, -1.098203, 1.570796, 1.627416],accel_mss,speed_ms,0,blend_radius_m)
    movel([0.057494, -0.814021, -2.800281, -1.098086, 1.570796, 1.628290],accel_mss,speed_ms,0,blend_radius_m)
    movel([0.058529, -0.813854, -2.800310, -1.098225, 1.570796, 1.629325],accel_mss,speed_ms,0,blend_radius_m)
    movel([0.060034, -0.813131, -2.800435, -1.098823, 1.570796, 1.630831],accel_mss,speed_ms,0,blend_radius_m)
    movel([0.061620, -0.811965, -2.800636, -1.099788, 1.570796, 1.632416],accel_mss,speed_ms,0,blend_radius_m)
    movel([0.064797, -0.808885, -2.801164, -1.102340, 1.570796, 1.635593],accel_mss,speed_ms,0,blend_radius_m)
    movel([0.068276, -0.804979, -2.801826, -1.105584, 1.570796, 1.639072],accel_mss,speed_ms,0,blend_radius_m)
    movel([0.071601, -0.800913, -2.802506, -1.108970, 1.570796, 1.642398],accel_mss,speed_ms,0,blend_radius_m)
    movel([0.077924, -0.792402, -2.803904, -1.116084, 1.570796, 1.648720],accel_mss,speed_ms,0,blend_radius_m)
    movel([0.090261, -0.774677, -2.806696, -1.131016, 1.570796, 1.661058],accel_mss,speed_ms,0,blend_radius_m)
    movel([0.096359, -0.766367, -2.807952, -1.138070, 1.570796, 1.667156],accel_mss,speed_ms,0,blend_radius_m)
    movel([0.099948, -0.761844, -2.808622, -1.141924, 1.570796, 1.670745],accel_mss,speed_ms,0,blend_radius_m)
    movel([0.103577, -0.757735, -2.809221, -1.145433, 1.570796, 1.674373],accel_mss,speed_ms,0,blend_radius_m)
    movel([0.105330, -0.755988, -2.809474, -1.146927, 1.570796, 1.676126],accel_mss,speed_ms,0,blend_radius_m)
    movel([0.107002, -0.754532, -2.809683, -1.148174, 1.570796, 1.677799],accel_mss,speed_ms,0,blend_radius_m)
    movel([0.108558, -0.753429, -2.809841, -1.149119, 1.570796, 1.679355],accel_mss,speed_ms,0,blend_radius_m)
    movel([0.109969, -0.752746, -2.809938, -1.149704, 1.570796, 1.680766],accel_mss,speed_ms,0,blend_radius_m)
    movel([0.111199, -0.752542, -2.809967, -1.149880, 1.570796, 1.681995],accel_mss,speed_ms,0,blend_radius_m)
    movel([0.112220, -0.752875, -2.809920, -1.149594, 1.570796, 1.683017],accel_mss,speed_ms,0,blend_radius_m)
    movel([0.113001, -0.753814, -2.809786, -1.148789, 1.570796, 1.683797],accel_mss,speed_ms,0,blend_radius_m)
    movel([0.113504, -0.755418, -2.809556, -1.147415, 1.570796, 1.684301],accel_mss,speed_ms,0,blend_radius_m)
    movel([0.113900, -0.758692, -2.809082, -1.144615, 1.570796, 1.684696],accel_mss,speed_ms,0,blend_radius_m)
    movel([0.113933, -0.762170, -2.808574, -1.141645, 1.570796, 1.684729],accel_mss,speed_ms,0,blend_radius_m)
    movel([0.113628, -0.765825, -2.808033, -1.138531, 1.570796, 1.684425],accel_mss,speed_ms,0,blend_radius_m)
    movel([0.113010, -0.769643, -2.807461, -1.135285, 1.570796, 1.683806],accel_mss,speed_ms,0,blend_radius_m)
    movel([0.112094, -0.773592, -2.806862, -1.131934, 1.570796, 1.682890],accel_mss,speed_ms,0,blend_radius_m)
    movel([0.110904, -0.777657, -2.806238, -1.128494, 1.570796, 1.681700],accel_mss,speed_ms,0,blend_radius_m)
    movel([0.109458, -0.781819, -2.805590, -1.124980, 1.570796, 1.680255],accel_mss,speed_ms,0,blend_radius_m)
    movel([0.107781, -0.786057, -2.804921, -1.121411, 1.570796, 1.678577],accel_mss,speed_ms,0,blend_radius_m)
    movel([0.103808, -0.794677, -2.803534, -1.114178, 1.570796, 1.674604],accel_mss,speed_ms,0,blend_radius_m)
    movel([0.099134, -0.803382, -2.802094, -1.106913, 1.570796, 1.669930],accel_mss,speed_ms,0,blend_radius_m)
    movel([0.093902, -0.812037, -2.800624, -1.099728, 1.570796, 1.664698],accel_mss,speed_ms,0,blend_radius_m)
    movel([0.088264, -0.820509, -2.799147, -1.092733, 1.570796, 1.659060],accel_mss,speed_ms,0,blend_radius_m)
    movel([0.075359, -0.838936, -2.795802, -1.077651, 1.570796, 1.646155],accel_mss,speed_ms,0,blend_radius_m)
    movel([0.068603, -0.847869, -2.794113, -1.070407, 1.570796, 1.639399],accel_mss,speed_ms,0,blend_radius_m)
    movel([0.065167, -0.852056, -2.793306, -1.067027, 1.570796, 1.635963],accel_mss,speed_ms,0,blend_radius_m)
    movel([0.061694, -0.855984, -2.792540, -1.063864, 1.570796, 1.632490],accel_mss,speed_ms,0,blend_radius_m)
    movel([0.059437, -0.858325, -2.792080, -1.061984, 1.570796, 1.630233],accel_mss,speed_ms,0,blend_radius_m)
    movel([0.057179, -0.860444, -2.791660, -1.060285, 1.570796, 1.627975],accel_mss,speed_ms,0,blend_radius_m)
    movel([0.054933, -0.862311, -2.791288, -1.058790, 1.570796, 1.625729],accel_mss,speed_ms,0,blend_radius_m)
    movel([0.052717, -0.863888, -2.790973, -1.057528, 1.570796, 1.623513],accel_mss,speed_ms,0,blend_radius_m)
    movel([0.050553, -0.865143, -2.790721, -1.056525, 1.570796, 1.621349],accel_mss,speed_ms,0,blend_radius_m)
    movel([0.048453, -0.866043, -2.790539, -1.055807, 1.570796, 1.619249],accel_mss,speed_ms,0,blend_radius_m)
    movel([0.046439, -0.866544, -2.790438, -1.055407, 1.570796, 1.617235],accel_mss,speed_ms,0,blend_radius_m)
    movel([0.044523, -0.866615, -2.790424, -1.055351, 1.570796, 1.615319],accel_mss,speed_ms,0,blend_radius_m)
    movel([0.042794, -0.866215, -2.790504, -1.055670, 1.570796, 1.613590],accel_mss,speed_ms,0,blend_radius_m)
    movel([0.041359, -0.865430, -2.790663, -1.056296, 1.570796, 1.612156],accel_mss,speed_ms,0,blend_radius_m)
    movel([0.036556, -0.860980, -2.791554, -1.059855, 1.570796, 1.607353],accel_mss,speed_ms,0,blend_radius_m)
    movel([0.035080, -0.860188, -2.791711, -1.060490, 1.570796, 1.605876],accel_mss,speed_ms,0,blend_radius_m)
    movel([0.033287, -0.859792, -2.791790, -1.060808, 1.570796, 1.604083],accel_mss,speed_ms,0,blend_radius_m)
    movel([0.032466, -0.859929, -2.791762, -1.060698, 1.570796, 1.603262],accel_mss,speed_ms,0,blend_radius_m)
    movel([0.032082, -0.860470, -2.791655, -1.060264, 1.570796, 1.602878],accel_mss,speed_ms,0,blend_radius_m)
    movel([0.031576, -0.861697, -2.791411, -1.059281, 1.570796, 1.602373],accel_mss,speed_ms,0,blend_radius_m)
    movel([0.030256, -0.865852, -2.790578, -1.055960, 1.570796, 1.601052],accel_mss,speed_ms,0,blend_radius_m)
    movel([0.026967, -0.878211, -2.788040, -1.046138, 1.570796, 1.597764],accel_mss,speed_ms,0,blend_radius_m)
    movel([0.021878, -0.898547, -2.783667, -1.030175, 1.570796, 1.592674],accel_mss,speed_ms,0,blend_radius_m)
    movel([0.018226, -0.909445, -2.781220, -1.021725, 1.570796, 1.589022],accel_mss,speed_ms,0,blend_radius_m)
    movel([0.014190, -0.920310, -2.778705, -1.013374, 1.570796, 1.584987],accel_mss,speed_ms,0,blend_radius_m)
    movel([0.009825, -0.931110, -2.776131, -1.005148, 1.570796, 1.580621],accel_mss,speed_ms,0,blend_radius_m)
    movel([0.005197, -0.941800, -2.773508, -0.997081, 1.570796, 1.575993],accel_mss,speed_ms,0,blend_radius_m)
    movel([-0.000923, -0.955304, -2.770085, -0.987000, 1.570796, 1.569874],accel_mss,speed_ms,0,blend_radius_m)
    movel([-0.007205, -0.968630, -2.766585, -0.977174, 1.570796, 1.563592],accel_mss,speed_ms,0,blend_radius_m)
    movel([-0.013697, -0.981730, -2.763022, -0.967637, 1.570796, 1.557100],accel_mss,speed_ms,0,blend_radius_m)
    movel([-0.020459, -0.994561, -2.759412, -0.958415, 1.570796, 1.550338],accel_mss,speed_ms,0,blend_radius_m)
    movel([-0.027538, -1.007076, -2.755774, -0.949538, 1.570796, 1.543258],accel_mss,speed_ms,0,blend_radius_m)
    movel([-0.031209, -1.013203, -2.753950, -0.945236, 1.570796, 1.539587],accel_mss,speed_ms,0,blend_radius_m)
    movel([-0.034982, -1.019241, -2.752124, -0.941024, 1.570796, 1.535814],accel_mss,speed_ms,0,blend_radius_m)
    movel([-0.038862, -1.025183, -2.750299, -0.936907, 1.570796, 1.531934],accel_mss,speed_ms,0,blend_radius_m)
    movel([-0.042852, -1.031023, -2.748479, -0.932887, 1.570796, 1.527944],accel_mss,speed_ms,0,blend_radius_m)
    movel([-0.046959, -1.036763, -2.746663, -0.928963, 1.570796, 1.523837],accel_mss,speed_ms,0,blend_radius_m)
    movel([-0.051195, -1.042396, -2.744855, -0.925138, 1.570796, 1.519601],accel_mss,speed_ms,0,blend_radius_m)
    movel([-0.056371, -1.048939, -2.742723, -0.920727, 1.570796, 1.514425],accel_mss,speed_ms,0,blend_radius_m)
    movel([-0.059066, -1.052085, -2.741685, -0.918619, 1.570796, 1.511730],accel_mss,speed_ms,0,blend_radius_m)
    movel([-0.063918, -1.057147, -2.739998, -0.915244, 1.570796, 1.506879],accel_mss,speed_ms,0,blend_radius_m)
    movel([-0.066429, -1.059462, -2.739220, -0.913707, 1.570796, 1.504367],accel_mss,speed_ms,0,blend_radius_m)
    movel([-0.068956, -1.061324, -2.738590, -0.912475, 1.570796, 1.501841],accel_mss,speed_ms,0,blend_radius_m)
    movel([-0.070084, -1.061863, -2.738407, -0.912119, 1.570796, 1.500713],accel_mss,speed_ms,0,blend_radius_m)
    movel([-0.071054, -1.062029, -2.738351, -0.912009, 1.570796, 1.499743],accel_mss,speed_ms,0,blend_radius_m)
    movel([-0.070384, -1.059319, -2.739268, -0.913802, 1.570796, 1.500412],accel_mss,speed_ms,0,blend_radius_m)
    movel([-0.070085, -1.056758, -2.740129, -0.915502, 1.570796, 1.500712],accel_mss,speed_ms,0,blend_radius_m)
    movel([-0.070167, -1.055657, -2.740497, -0.916235, 1.570796, 1.500629],accel_mss,speed_ms,0,blend_radius_m)
    movel([-0.070455, -1.054744, -2.740802, -0.916843, 1.570796, 1.500341],accel_mss,speed_ms,0,blend_radius_m)
    movel([-0.070984, -1.054065, -2.741028, -0.917296, 1.570796, 1.499812],accel_mss,speed_ms,0,blend_radius_m)
    movel([-0.071800, -1.053680, -2.741156, -0.917553, 1.570796, 1.498996],accel_mss,speed_ms,0,blend_radius_m)
    movel([-0.074299, -1.053501, -2.741216, -0.917672, 1.570796, 1.496497],accel_mss,speed_ms,0,blend_radius_m)
    movel([-0.074995, -1.053160, -2.741329, -0.917900, 1.570796, 1.495802],accel_mss,speed_ms,0,blend_radius_m)
    movel([-0.075477, -1.052592, -2.741518, -0.918280, 1.570796, 1.495319],accel_mss,speed_ms,0,blend_radius_m)
    movel([-0.075891, -1.050918, -2.742071, -0.919400, 1.570796, 1.494905],accel_mss,speed_ms,0,blend_radius_m)
    movel([-0.075764, -1.048777, -2.742776, -0.920836, 1.570796, 1.495032],accel_mss,speed_ms,0,blend_radius_m)
    movel([-0.075312, -1.046476, -2.743530, -0.922383, 1.570796, 1.495484],accel_mss,speed_ms,0,blend_radius_m)
    movel([-0.073518, -1.039374, -2.745828, -0.927186, 1.570796, 1.497279],accel_mss,speed_ms,0,blend_radius_m)
    movel([-0.071298, -1.032017, -2.748166, -0.932205, 1.570796, 1.499499],accel_mss,speed_ms,0,blend_radius_m)
    movel([-0.069956, -1.028258, -2.749344, -0.934787, 1.570796, 1.500841],accel_mss,speed_ms,0,blend_radius_m)
    movel([-0.068425, -1.024449, -2.750526, -0.937414, 1.570796, 1.502371],accel_mss,speed_ms,0,blend_radius_m)
    movel([-0.066676, -1.020600, -2.751709, -0.940080, 1.570796, 1.504121],accel_mss,speed_ms,0,blend_radius_m)
    movel([-0.064677, -1.016712, -2.752892, -0.942785, 1.570796, 1.506120],accel_mss,speed_ms,0,blend_radius_m)
    movel([-0.062393, -1.012948, -2.754027, -0.945415, 1.570796, 1.508403],accel_mss,speed_ms,0,blend_radius_m)
    movel([-0.054713, -1.002033, -2.757255, -0.953102, 1.570796, 1.516083],accel_mss,speed_ms,0,blend_radius_m)
    movel([-0.048747, -0.992549, -2.759987, -0.959853, 1.570796, 1.522049],accel_mss,speed_ms,0,blend_radius_m)
    movel([-0.042918, -0.982852, -2.762711, -0.966825, 1.570796, 1.527878],accel_mss,speed_ms,0,blend_radius_m)
    movel([-0.040332, -0.978431, -2.763931, -0.970027, 1.570796, 1.530464],accel_mss,speed_ms,0,blend_radius_m)
    speed_ms = 0.005
    movel([-0.040332, -0.968607, -2.758169, -0.985613, 1.570796, 1.530464],accel_mss,speed_ms,0,blend_radius_m)
    speed_ms = 0.040
    movel([-0.093122, -1.046614, -2.734729, -0.931046, 1.570796, 1.477674],accel_mss,speed_ms,0,blend_radius_m)
    speed_ms = 0.005
    movel([-0.093122, -1.056630, -2.740172, -0.915587, 1.570796, 1.477674],accel_mss,speed_ms,0,blend_radius_m)
    speed_ms = 0.025
    movel([-0.088514, -1.059684, -2.739145, -0.913560, 1.570796, 1.482283],accel_mss,speed_ms,0,blend_radius_m)
    movel([-0.086238, -1.061524, -2.738522, -0.912343, 1.570796, 1.484558],accel_mss,speed_ms,0,blend_radius_m)
    movel([-0.084156, -1.063620, -2.737810, -0.910959, 1.570796, 1.486640],accel_mss,speed_ms,0,blend_radius_m)
    movel([-0.082385, -1.065989, -2.737000, -0.909400, 1.570796, 1.488411],accel_mss,speed_ms,0,blend_radius_m)
    movel([-0.081051, -1.068655, -2.736083, -0.907651, 1.570796, 1.489746],accel_mss,speed_ms,0,blend_radius_m)
    movel([-0.080272, -1.071644, -2.735047, -0.905698, 1.570796, 1.490524],accel_mss,speed_ms,0,blend_radius_m)
    movel([-0.080130, -1.073269, -2.734481, -0.904639, 1.570796, 1.490666],accel_mss,speed_ms,0,blend_radius_m)
    movel([-0.080171, -1.074978, -2.733883, -0.903528, 1.570796, 1.490625],accel_mss,speed_ms,0,blend_radius_m)
    movel([-0.081282, -1.074682, -2.733987, -0.903720, 1.570796, 1.489514],accel_mss,speed_ms,0,blend_radius_m)
    movel([-0.082008, -1.074088, -2.734195, -0.904106, 1.570796, 1.488789],accel_mss,speed_ms,0,blend_radius_m)
    movel([-0.083540, -1.072660, -2.734693, -0.905035, 1.570796, 1.487256],accel_mss,speed_ms,0,blend_radius_m)
    movel([-0.085642, -1.071670, -2.735038, -0.905681, 1.570796, 1.485155],accel_mss,speed_ms,0,blend_radius_m)
    movel([-0.087960, -1.070971, -2.735281, -0.906137, 1.570796, 1.482836],accel_mss,speed_ms,0,blend_radius_m)
    movel([-0.090469, -1.070549, -2.735428, -0.906412, 1.570796, 1.480327],accel_mss,speed_ms,0,blend_radius_m)
    movel([-0.093141, -1.070399, -2.735480, -0.906511, 1.570796, 1.477655],accel_mss,speed_ms,0,blend_radius_m)
    movel([-0.095950, -1.070506, -2.735442, -0.906440, 1.570796, 1.474847],accel_mss,speed_ms,0,blend_radius_m)
    movel([-0.098866, -1.070865, -2.735318, -0.906206, 1.570796, 1.471931],accel_mss,speed_ms,0,blend_radius_m)
    movel([-0.101865, -1.071465, -2.735110, -0.905814, 1.570796, 1.468931],accel_mss,speed_ms,0,blend_radius_m)
    movel([-0.104918, -1.072290, -2.734823, -0.905276, 1.570796, 1.465879],accel_mss,speed_ms,0,blend_radius_m)
    movel([-0.106974, -1.073015, -2.734570, -0.904804, 1.570796, 1.463823],accel_mss,speed_ms,0,blend_radius_m)
    movel([-0.108597, -1.073795, -2.734297, -0.904297, 1.570796, 1.462200],accel_mss,speed_ms,0,blend_radius_m)
    movel([-0.109819, -1.074617, -2.734010, -0.903762, 1.570796, 1.460977],accel_mss,speed_ms,0,blend_radius_m)
    movel([-0.110677, -1.075472, -2.733710, -0.903207, 1.570796, 1.460119],accel_mss,speed_ms,0,blend_radius_m)
    movel([-0.111210, -1.076357, -2.733399, -0.902633, 1.570796, 1.459587],accel_mss,speed_ms,0,blend_radius_m)
    movel([-0.111450, -1.077263, -2.733080, -0.902046, 1.570796, 1.459346],accel_mss,speed_ms,0,blend_radius_m)
    movel([-0.111443, -1.078186, -2.732754, -0.901449, 1.570796, 1.459353],accel_mss,speed_ms,0,blend_radius_m)
    movel([-0.111217, -1.079115, -2.732425, -0.900848, 1.570796, 1.459579],accel_mss,speed_ms,0,blend_radius_m)
    movel([-0.110274, -1.080979, -2.731764, -0.899646, 1.570796, 1.460522],accel_mss,speed_ms,0,blend_radius_m)
    movel([-0.106117, -1.086175, -2.729903, -0.896311, 1.570796, 1.464679],accel_mss,speed_ms,0,blend_radius_m)
    movel([-0.108813, -1.085296, -2.730219, -0.896874, 1.570796, 1.461983],accel_mss,speed_ms,0,blend_radius_m)
    movel([-0.114098, -1.083404, -2.730898, -0.898087, 1.570796, 1.456698],accel_mss,speed_ms,0,blend_radius_m)
    movel([-0.117064, -1.082969, -2.731054, -0.898366, 1.570796, 1.453732],accel_mss,speed_ms,0,blend_radius_m)
    movel([-0.120621, -1.082985, -2.731048, -0.898356, 1.570796, 1.450175],accel_mss,speed_ms,0,blend_radius_m)
    movel([-0.124303, -1.083224, -2.730962, -0.898202, 1.570796, 1.446493],accel_mss,speed_ms,0,blend_radius_m)
    movel([-0.131751, -1.083884, -2.730726, -0.897779, 1.570796, 1.439045],accel_mss,speed_ms,0,blend_radius_m)
    movel([-0.135375, -1.084063, -2.730662, -0.897664, 1.570796, 1.435422],accel_mss,speed_ms,0,blend_radius_m)
    movel([-0.138835, -1.083980, -2.730692, -0.897717, 1.570796, 1.431961],accel_mss,speed_ms,0,blend_radius_m)
    movel([-0.142064, -1.083520, -2.730857, -0.898013, 1.570796, 1.428732],accel_mss,speed_ms,0,blend_radius_m)
    movel([-0.144994, -1.082554, -2.731202, -0.898633, 1.570796, 1.425802],accel_mss,speed_ms,0,blend_radius_m)
    movel([-0.142066, -1.087156, -2.729549, -0.895684, 1.570796, 1.428730],accel_mss,speed_ms,0,blend_radius_m)
    movel([-0.140408, -1.089371, -2.728746, -0.894271, 1.570796, 1.430388],accel_mss,speed_ms,0,blend_radius_m)
    movel([-0.138560, -1.091112, -2.728113, -0.893165, 1.570796, 1.432236],accel_mss,speed_ms,0,blend_radius_m)
    movel([-0.141511, -1.090277, -2.728417, -0.893695, 1.570796, 1.429285],accel_mss,speed_ms,0,blend_radius_m)
    movel([-0.144714, -1.089835, -2.728578, -0.893977, 1.570796, 1.426083],accel_mss,speed_ms,0,blend_radius_m)
    movel([-0.151368, -1.089350, -2.728754, -0.894285, 1.570796, 1.419428],accel_mss,speed_ms,0,blend_radius_m)
    movel([-0.153487, -1.089001, -2.728881, -0.894508, 1.570796, 1.417310],accel_mss,speed_ms,0,blend_radius_m)
    movel([-0.155390, -1.088415, -2.729093, -0.894881, 1.570796, 1.415406],accel_mss,speed_ms,0,blend_radius_m)
    movel([-0.158780, -1.086768, -2.729689, -0.895932, 1.570796, 1.412016],accel_mss,speed_ms,0,blend_radius_m)
    movel([-0.162022, -1.084900, -2.730362, -0.897128, 1.570796, 1.408775],accel_mss,speed_ms,0,blend_radius_m)
    movel([-0.165594, -1.083320, -2.730928, -0.898141, 1.570796, 1.405202],accel_mss,speed_ms,0,blend_radius_m)
    movel([-0.166857, -1.083009, -2.731039, -0.898340, 1.570796, 1.403939],accel_mss,speed_ms,0,blend_radius_m)
    movel([-0.168262, -1.082943, -2.731063, -0.898383, 1.570796, 1.402535],accel_mss,speed_ms,0,blend_radius_m)
    movel([-0.169781, -1.083276, -2.730944, -0.898169, 1.570796, 1.401015],accel_mss,speed_ms,0,blend_radius_m)
    movel([-0.170570, -1.083631, -2.730817, -0.897941, 1.570796, 1.400227],accel_mss,speed_ms,0,blend_radius_m)
    movel([-0.171376, -1.084146, -2.730632, -0.897610, 1.570796, 1.399420],accel_mss,speed_ms,0,blend_radius_m)
    movel([-0.172224, -1.084860, -2.730376, -0.897153, 1.570796, 1.398572],accel_mss,speed_ms,0,blend_radius_m)
    movel([-0.172969, -1.085668, -2.730085, -0.896636, 1.570796, 1.397828],accel_mss,speed_ms,0,blend_radius_m)
    movel([-0.174198, -1.087493, -2.729427, -0.895469, 1.570796, 1.396598],accel_mss,speed_ms,0,blend_radius_m)
    movel([-0.175125, -1.089452, -2.728717, -0.894220, 1.570796, 1.395671],accel_mss,speed_ms,0,blend_radius_m)
    movel([-0.175812, -1.091378, -2.728015, -0.892996, 1.570796, 1.394984],accel_mss,speed_ms,0,blend_radius_m)
    movel([-0.176919, -1.089059, -2.728860, -0.894471, 1.570796, 1.393878],accel_mss,speed_ms,0,blend_radius_m)
    movel([-0.178255, -1.086993, -2.729607, -0.895788, 1.570796, 1.392542],accel_mss,speed_ms,0,blend_radius_m)
    movel([-0.181370, -1.083368, -2.730911, -0.898110, 1.570796, 1.389427],accel_mss,speed_ms,0,blend_radius_m)
    movel([-0.184663, -1.079933, -2.732135, -0.900320, 1.570796, 1.386133],accel_mss,speed_ms,0,blend_radius_m)
    movel([-0.187634, -1.076100, -2.733489, -0.902800, 1.570796, 1.383162],accel_mss,speed_ms,0,blend_radius_m)
    movel([-0.188493, -1.074334, -2.734109, -0.903946, 1.570796, 1.382303],accel_mss,speed_ms,0,blend_radius_m)
    movel([-0.189079, -1.072280, -2.734826, -0.905283, 1.570796, 1.381718],accel_mss,speed_ms,0,blend_radius_m)
    movel([-0.189428, -1.069994, -2.735620, -0.906775, 1.570796, 1.381368],accel_mss,speed_ms,0,blend_radius_m)
    movel([-0.189583, -1.067539, -2.736468, -0.908383, 1.570796, 1.381213],accel_mss,speed_ms,0,blend_radius_m)
    movel([-0.189440, -1.062334, -2.738247, -0.911808, 1.570796, 1.381356],accel_mss,speed_ms,0,blend_radius_m)
    movel([-0.188953, -1.057150, -2.739998, -0.915242, 1.570796, 1.381843],accel_mss,speed_ms,0,blend_radius_m)
    speed_ms = 0.005
    movel([-0.188953, -1.047133, -2.734557, -0.930698, 1.570796, 1.381843],accel_mss,speed_ms,0,blend_radius_m)
    speed_ms = 0.040
    # Splitting Linear movement in 2 (instruction 806: MoveL 765)
    movel([-0.160518, -0.969003, -2.758061, -0.985324, 1.570796, 1.410279],accel_mss,speed_ms,0,blend_radius_m)
    movel([-0.127076, -0.880602, -2.779460, -1.052327, 1.570796, 1.443720],accel_mss,speed_ms,0,blend_radius_m)
    speed_ms = 0.005
    movel([-0.127076, -0.889934, -2.785550, -1.036906, 1.570796, 1.443720],accel_mss,speed_ms,0,blend_radius_m)
    speed_ms = 0.025
    movel([-0.129184, -0.892633, -2.784964, -1.034792, 1.570796, 1.441613],accel_mss,speed_ms,0,blend_radius_m)
    movel([-0.129327, -0.893070, -2.784869, -1.034450, 1.570796, 1.441470],accel_mss,speed_ms,0,blend_radius_m)
    movel([-0.129124, -0.893540, -2.784767, -1.034082, 1.570796, 1.441672],accel_mss,speed_ms,0,blend_radius_m)
    movel([-0.127771, -0.894592, -2.784537, -1.033260, 1.570796, 1.443025],accel_mss,speed_ms,0,blend_radius_m)
    movel([-0.121910, -0.897073, -2.783992, -1.031324, 1.570796, 1.448886],accel_mss,speed_ms,0,blend_radius_m)
    movel([-0.113033, -0.899954, -2.783355, -1.029080, 1.570796, 1.457763],accel_mss,speed_ms,0,blend_radius_m)
    movel([-0.102546, -0.903091, -2.782655, -1.026643, 1.570796, 1.468250],accel_mss,speed_ms,0,blend_radius_m)
    movel([-0.082100, -0.909176, -2.781281, -1.021933, 1.570796, 1.488696],accel_mss,speed_ms,0,blend_radius_m)
    movel([-0.070616, -0.912545, -2.780510, -1.019334, 1.570796, 1.500180],accel_mss,speed_ms,0,blend_radius_m)
    movel([-0.069504, -0.912687, -2.780477, -1.019225, 1.570796, 1.501292],accel_mss,speed_ms,0,blend_radius_m)
    movel([-0.068251, -0.912558, -2.780507, -1.019325, 1.570796, 1.502546],accel_mss,speed_ms,0,blend_radius_m)
    movel([-0.066940, -0.912001, -2.780635, -1.019754, 1.570796, 1.503856],accel_mss,speed_ms,0,blend_radius_m)
    movel([-0.066285, -0.911515, -2.780746, -1.020128, 1.570796, 1.504511],accel_mss,speed_ms,0,blend_radius_m)
    movel([-0.065647, -0.910861, -2.780896, -1.020632, 1.570796, 1.505150],accel_mss,speed_ms,0,blend_radius_m)
    movel([-0.064726, -0.909465, -2.781215, -1.021709, 1.570796, 1.506070],accel_mss,speed_ms,0,blend_radius_m)
    movel([-0.064072, -0.908014, -2.781545, -1.022830, 1.570796, 1.506725],accel_mss,speed_ms,0,blend_radius_m)
    movel([-0.061077, -0.899977, -2.783350, -1.029062, 1.570796, 1.509719],accel_mss,speed_ms,0,blend_radius_m)
    movel([-0.058603, -0.892029, -2.785096, -1.035265, 1.570796, 1.512193],accel_mss,speed_ms,0,blend_radius_m)
    movel([-0.056631, -0.884206, -2.786777, -1.041406, 1.570796, 1.514166],accel_mss,speed_ms,0,blend_radius_m)
    movel([-0.055120, -0.876537, -2.788389, -1.047463, 1.570796, 1.515677],accel_mss,speed_ms,0,blend_radius_m)
    movel([-0.054047, -0.869052, -2.789929, -1.053408, 1.570796, 1.516750],accel_mss,speed_ms,0,blend_radius_m)
    movel([-0.053374, -0.861779, -2.791395, -1.059216, 1.570796, 1.517422],accel_mss,speed_ms,0,blend_radius_m)
    movel([-0.053071, -0.854749, -2.792782, -1.064858, 1.570796, 1.517725],accel_mss,speed_ms,0,blend_radius_m)
    movel([-0.053102, -0.847998, -2.794088, -1.070302, 1.570796, 1.517694],accel_mss,speed_ms,0,blend_radius_m)
    movel([-0.053330, -0.845081, -2.794645, -1.072664, 1.570796, 1.517466],accel_mss,speed_ms,0,blend_radius_m)
    movel([-0.053831, -0.842569, -2.795120, -1.074700, 1.570796, 1.516965],accel_mss,speed_ms,0,blend_radius_m)
    movel([-0.054603, -0.840459, -2.795517, -1.076413, 1.570796, 1.516193],accel_mss,speed_ms,0,blend_radius_m)
    movel([-0.055630, -0.838738, -2.795839, -1.077813, 1.570796, 1.515167],accel_mss,speed_ms,0,blend_radius_m)
    movel([-0.056906, -0.837404, -2.796087, -1.078899, 1.570796, 1.513890],accel_mss,speed_ms,0,blend_radius_m)
    movel([-0.058424, -0.836452, -2.796263, -1.079674, 1.570796, 1.512372],accel_mss,speed_ms,0,blend_radius_m)
    movel([-0.060169, -0.835862, -2.796372, -1.080155, 1.570796, 1.510627],accel_mss,speed_ms,0,blend_radius_m)
    movel([-0.062137, -0.835630, -2.796415, -1.080344, 1.570796, 1.508659],accel_mss,speed_ms,0,blend_radius_m)
    movel([-0.064312, -0.835746, -2.796394, -1.080249, 1.570796, 1.506485],accel_mss,speed_ms,0,blend_radius_m)
    movel([-0.066683, -0.836198, -2.796310, -1.079880, 1.570796, 1.504114],accel_mss,speed_ms,0,blend_radius_m)
    movel([-0.069245, -0.836975, -2.796166, -1.079248, 1.570796, 1.501552],accel_mss,speed_ms,0,blend_radius_m)
    movel([-0.071976, -0.838064, -2.795964, -1.078361, 1.570796, 1.498820],accel_mss,speed_ms,0,blend_radius_m)
    movel([-0.077923, -0.841133, -2.795390, -1.075866, 1.570796, 1.492874],accel_mss,speed_ms,0,blend_radius_m)
    movel([-0.084421, -0.845296, -2.794604, -1.072489, 1.570796, 1.486375],accel_mss,speed_ms,0,blend_radius_m)
    movel([-0.090248, -0.849687, -2.793764, -1.068938, 1.570796, 1.480548],accel_mss,speed_ms,0,blend_radius_m)
    movel([-0.095935, -0.854599, -2.792811, -1.064978, 1.570796, 1.474861],accel_mss,speed_ms,0,blend_radius_m)
    movel([-0.101486, -0.859952, -2.791758, -1.060679, 1.570796, 1.469311],accel_mss,speed_ms,0,blend_radius_m)
    movel([-0.106894, -0.865641, -2.790620, -1.056128, 1.570796, 1.463903],accel_mss,speed_ms,0,blend_radius_m)
    movel([-0.112150, -0.871568, -2.789415, -1.051406, 1.570796, 1.458646],accel_mss,speed_ms,0,blend_radius_m)
    movel([-0.117267, -0.877651, -2.788157, -1.046581, 1.570796, 1.453529],accel_mss,speed_ms,0,blend_radius_m)
    movel([-0.127076, -0.889934, -2.785550, -1.036906, 1.570796, 1.443720],accel_mss,speed_ms,0,blend_radius_m)
    movel([-0.129184, -0.892633, -2.784964, -1.034792, 1.570796, 1.441613],accel_mss,speed_ms,0,blend_radius_m)
    movel([-0.129327, -0.893070, -2.784869, -1.034450, 1.570796, 1.441470],accel_mss,speed_ms,0,blend_radius_m)
    movel([-0.129124, -0.893540, -2.784767, -1.034082, 1.570796, 1.441672],accel_mss,speed_ms,0,blend_radius_m)
    movel([-0.128696, -0.893875, -2.784694, -1.033820, 1.570796, 1.442100],accel_mss,speed_ms,0,blend_radius_m)
    speed_ms = 0.005
    movel([-0.128696, -0.884515, -2.778617, -1.049257, 1.570796, 1.442100],accel_mss,speed_ms,0,blend_radius_m)
    speed_ms = 0.040
    movel([-0.148208, -0.861864, -2.783366, -1.067159, 1.570796, 1.422589],accel_mss,speed_ms,0,blend_radius_m)
    speed_ms = 0.005
    movel([-0.148208, -0.871052, -2.789521, -1.051816, 1.570796, 1.422589],accel_mss,speed_ms,0,blend_radius_m)
    speed_ms = 0.025
    movel([-0.148572, -0.868567, -2.790028, -1.053794, 1.570796, 1.422224],accel_mss,speed_ms,0,blend_radius_m)
    movel([-0.149389, -0.866479, -2.790451, -1.055459, 1.570796, 1.421407],accel_mss,speed_ms,0,blend_radius_m)
    movel([-0.150642, -0.864844, -2.790781, -1.056764, 1.570796, 1.420154],accel_mss,speed_ms,0,blend_radius_m)
    movel([-0.152301, -0.863700, -2.791011, -1.057679, 1.570796, 1.418496],accel_mss,speed_ms,0,blend_radius_m)
    movel([-0.157266, -0.862132, -2.791324, -1.058933, 1.570796, 1.413531],accel_mss,speed_ms,0,blend_radius_m)
    movel([-0.158495, -0.861438, -2.791463, -1.059489, 1.570796, 1.412302],accel_mss,speed_ms,0,blend_radius_m)
    movel([-0.159388, -0.860503, -2.791649, -1.060238, 1.570796, 1.411408],accel_mss,speed_ms,0,blend_radius_m)
    movel([-0.159787, -0.859275, -2.791892, -1.061222, 1.570796, 1.411010],accel_mss,speed_ms,0,blend_radius_m)
    movel([-0.159519, -0.857684, -2.792206, -1.062499, 1.570796, 1.411277],accel_mss,speed_ms,0,blend_radius_m)
    movel([-0.158496, -0.855627, -2.792610, -1.064152, 1.570796, 1.412300],accel_mss,speed_ms,0,blend_radius_m)
    movel([-0.157173, -0.854007, -2.792927, -1.065455, 1.570796, 1.413623],accel_mss,speed_ms,0,blend_radius_m)
    movel([-0.155636, -0.852773, -2.793167, -1.066449, 1.570796, 1.415161],accel_mss,speed_ms,0,blend_radius_m)
    movel([-0.153982, -0.851875, -2.793341, -1.067172, 1.570796, 1.416814],accel_mss,speed_ms,0,blend_radius_m)
    movel([-0.150724, -0.850900, -2.793530, -1.067959, 1.570796, 1.420072],accel_mss,speed_ms,0,blend_radius_m)
    movel([-0.148143, -0.850668, -2.793575, -1.068146, 1.570796, 1.422653],accel_mss,speed_ms,0,blend_radius_m)
    movel([-0.149321, -0.848135, -2.794062, -1.070192, 1.570796, 1.421476],accel_mss,speed_ms,0,blend_radius_m)
    movel([-0.151025, -0.846251, -2.794422, -1.071716, 1.570796, 1.419772],accel_mss,speed_ms,0,blend_radius_m)
    movel([-0.155392, -0.843635, -2.794919, -1.073835, 1.570796, 1.415404],accel_mss,speed_ms,0,blend_radius_m)
    movel([-0.159988, -0.841179, -2.795382, -1.075828, 1.570796, 1.410808],accel_mss,speed_ms,0,blend_radius_m)
    movel([-0.161984, -0.839490, -2.795698, -1.077201, 1.570796, 1.408813],accel_mss,speed_ms,0,blend_radius_m)
    movel([-0.163557, -0.837206, -2.796124, -1.079060, 1.570796, 1.407239],accel_mss,speed_ms,0,blend_radius_m)
    movel([-0.164261, -0.835458, -2.796447, -1.080484, 1.570796, 1.406535],accel_mss,speed_ms,0,blend_radius_m)
    movel([-0.164602, -0.833827, -2.796748, -1.081815, 1.570796, 1.406195],accel_mss,speed_ms,0,blend_radius_m)
    movel([-0.164612, -0.832318, -2.797024, -1.083047, 1.570796, 1.406184],accel_mss,speed_ms,0,blend_radius_m)
    movel([-0.164323, -0.830942, -2.797275, -1.084171, 1.570796, 1.406473],accel_mss,speed_ms,0,blend_radius_m)
    movel([-0.163779, -0.829715, -2.797499, -1.085176, 1.570796, 1.407017],accel_mss,speed_ms,0,blend_radius_m)
    movel([-0.163009, -0.828631, -2.797695, -1.086063, 1.570796, 1.407787],accel_mss,speed_ms,0,blend_radius_m)
    movel([-0.162059, -0.827711, -2.797861, -1.086817, 1.570796, 1.408737],accel_mss,speed_ms,0,blend_radius_m)
    movel([-0.160956, -0.826959, -2.797997, -1.087433, 1.570796, 1.409840],accel_mss,speed_ms,0,blend_radius_m)
    movel([-0.159743, -0.826388, -2.798099, -1.087901, 1.570796, 1.411053],accel_mss,speed_ms,0,blend_radius_m)
    movel([-0.158463, -0.826010, -2.798167, -1.088211, 1.570796, 1.412333],accel_mss,speed_ms,0,blend_radius_m)
    movel([-0.155834, -0.825858, -2.798195, -1.088336, 1.570796, 1.414963],accel_mss,speed_ms,0,blend_radius_m)
